// Verwendung der Presets: {attribute 'Preset.HochlaufzeitMin' := '@.tMinZeit'}
// oder dirket als Zahl: {attribute 'Preset.HochlaufzeitMin' := 'T#1M'}
// muss über der Instanz von ST_UniAntrAnstgParamAggrHF stehen
// mögliche Presets: 'Preset.HochlaufzeitMin', 'Preset.HochlaufzeitMax'
{attribute 'MaschPara.Margin' := '0 10 0 0'}	
{attribute 'MaschPara.Name' := 'Hochlaufphase 1 Zeit'}
{attribute 'MaschPara.Type' := 'min'}
{attribute 'MaschPara.Min' := 'Preset.HochlaufzeitMin'}
{attribute 'MaschPara.Max' := 'Preset.HochlaufzeitMax'}
{attribute 'MaschPara.Info' := 'Minuten je Hochlaufphase mit der Drehzahl aus fBetrZyklDrehz1'}
{attribute 'MaschPara.TreeViewLayer' := '-1'}
{attribute 'MaschPara.GroupName' := 'Preset.GroupName'}
	tBetrZyklPhase1	:TIME	:= T#1M;
// Verwendung der Presets: {attribute 'Preset.HochlaufzeitMin' := '@.tMinZeit'}
// oder dirket als Zahl: {attribute 'Preset.HochlaufzeitMin' := 'T#1M'}
// muss über der Instanz von ST_UniAntrAnstgParamAggrHF stehen
// mögliche Presets: 'Preset.HochlaufzeitMin', 'Preset.HochlaufzeitMax'
{attribute 'MaschPara.Name' := 'Hochlaufphase 2 Zeit'}
{attribute 'MaschPara.Type' := 'min'}
{attribute 'MaschPara.Min' := 'Preset.HochlaufzeitMin'}
{attribute 'MaschPara.Max' := 'Preset.HochlaufzeitMax'}
{attribute 'MaschPara.Info' := 'Minuten je Hochlaufphase mit der Drehzahl aus fBetrZyklDrehz2'}
{attribute 'MaschPara.TreeViewLayer' := '-1'}
{attribute 'MaschPara.GroupName' := 'Preset.GroupName'}
	tBetrZyklPhase2	:TIME	:= T#1M;
// Verwendung der Presets: {attribute 'Preset.HochlaufzeitMin' := '@.tMinZeit'}
// oder dirket als Zahl: {attribute 'Preset.HochlaufzeitMin' := 'T#1M'}
// muss über der Instanz von ST_UniAntrAnstgParamAggrHF stehen
// mögliche Presets: 'Preset.HochlaufzeitMin', 'Preset.HochlaufzeitMax'
{attribute 'MaschPara.Name' := 'Hochlaufphase 3 Zeit'}
{attribute 'MaschPara.Type' := 'min'}
{attribute 'MaschPara.Min' := 'Preset.HochlaufzeitMin'}
{attribute 'MaschPara.Max' := 'Preset.HochlaufzeitMax'}
{attribute 'MaschPara.Info' := 'Minuten je Hochlaufphase mit der Drehzahl aus fBetrZyklDrehz3'}
{attribute 'MaschPara.TreeViewLayer' := '-1'}
{attribute 'MaschPara.GroupName' := 'Preset.GroupName'}
	tBetrZyklPhase3	:TIME	:= T#1M;
// Verwendung der Presets: {attribute 'Preset.HochlaufzeitMin' := '@.tMinZeit'}
// oder dirket als Zahl: {attribute 'Preset.HochlaufzeitMin' := 'T#1M'}
// muss über der Instanz von ST_UniAntrAnstgParamAggrHF stehen
// mögliche Presets: 'Preset.HochlaufzeitMin', 'Preset.HochlaufzeitMax'
{attribute 'MaschPara.Name' := 'Hochlaufphase 4 Zeit'}
{attribute 'MaschPara.Type' := 'min'}
{attribute 'MaschPara.Min' := 'Preset.HochlaufzeitMin'}
{attribute 'MaschPara.Max' := 'Preset.HochlaufzeitMax'}
{attribute 'MaschPara.Info' := 'Minuten je Hochlaufphase mit der Drehzahl aus fBetrZyklDrehz4'}
{attribute 'MaschPara.TreeViewLayer' := '-1'}
{attribute 'MaschPara.GroupName' := 'Preset.GroupName'}
	tBetrZyklPhase4	:TIME	:= T#1M;
// Verwendung der Presets: {attribute 'Preset.StillstandMin' := '@.tMinZeit'}
// oder dirket als Zahl: {attribute 'Preset.StillstandMin' := 'T#1M'}
// muss über der Instanz von ST_UniAntrAnstgParamAggrHF stehen
// mögliche Presets: 'Preset.StillstandMin', 'Preset.StillstandMax'
{attribute 'MaschPara.Name' := 'Maximale Stillstandzeit'}
{attribute 'MaschPara.Type' := 'min'}
{attribute 'MaschPara.Min' := 'Preset.StillstandMin'}
{attribute 'MaschPara.Max' := 'Preset.StillstandMax'}
{attribute 'MaschPara.Info' := 'Zeit in Minuten bis eine neue Hochlaufphase notwendig wird'}
{attribute 'MaschPara.TreeViewLayer' := '-1'}
{attribute 'MaschPara.GroupName' := 'Preset.GroupName'}
	tMaxStillstandszeit	:TIME	:= T#15M;
// Verwendung der Presets: {attribute 'Preset.HochlaufdrehzMin' := '@.fMinDrehzahl'}
// oder dirket als Zahl: {attribute 'Preset.HochlaufdrehzMin' := '50'}
// muss über der Instanz von ST_UniAntrAnstgParamAggrHF stehen
// mögliche Presets: 'Preset.HochlaufdrehzMin', 'Preset.HochlaufdrehzMax'
{attribute 'MaschPara.Name' := 'Hochlaufphase 1 Drehzahl'}
{attribute 'MaschPara.Type' := '%'}
{attribute 'MaschPara.Min' := 'Preset.HochlaufdrehzMin'}
{attribute 'MaschPara.Max' := 'Preset.HochlaufdrehzMax'}
{attribute 'MaschPara.Info' := 'Prozentuale Drehzahl je Hochlaufphase'}	
{attribute 'MaschPara.TreeViewLayer' := '-1'}
{attribute 'MaschPara.GroupName' := 'Preset.GroupName'}
	fBetrZyklDrehz1	:LREAL := 50;
// Verwendung der Presets: {attribute 'Preset.HochlaufdrehzMin' := '@.fMinDrehzahl'}
// oder dirket als Zahl: {attribute 'Preset.HochlaufdrehzMin' := '75'}
// muss über der Instanz von ST_UniAntrAnstgParamAggrHF stehen
// mögliche Presets: 'Preset.HochlaufdrehzMin', 'Preset.HochlaufdrehzMax'
{attribute 'MaschPara.Name' := 'Hochlaufphase 2 Drehzahl'}
{attribute 'MaschPara.Type' := '%'}
{attribute 'MaschPara.Min' := 'Preset.HochlaufdrehzMin'}
{attribute 'MaschPara.Max' := 'Preset.HochlaufdrehzMax'}
{attribute 'MaschPara.Info' := 'Prozentuale Drehzahl je Hochlaufphase'}	
{attribute 'MaschPara.TreeViewLayer' := '-1'}
{attribute 'MaschPara.GroupName' := 'Preset.GroupName'}
	fBetrZyklDrehz2	:LREAL := 75;
// Verwendung der Presets: {attribute 'Preset.HochlaufdrehzMin' := '@.fMinDrehzahl'}
// oder dirket als Zahl: {attribute 'Preset.HochlaufdrehzMin' := '100'}
// muss über der Instanz von ST_UniAntrAnstgParamAggrHF stehen
// mögliche Presets: 'Preset.HochlaufdrehzMin', 'Preset.HochlaufdrehzMax'
{attribute 'MaschPara.Name' := 'Hochlaufphase 3 Drehzahl'}
{attribute 'MaschPara.Type' := '%'}
{attribute 'MaschPara.Min' := 'Preset.HochlaufdrehzMin'}
{attribute 'MaschPara.Max' := 'Preset.HochlaufdrehzMax'}
{attribute 'MaschPara.Info' := 'Prozentuale Drehzahl je Hochlaufphase'}	
{attribute 'MaschPara.TreeViewLayer' := '-1'}
{attribute 'MaschPara.GroupName' := 'Preset.GroupName'}
	fBetrZyklDrehz3	:LREAL := 100;
// Verwendung der Presets: {attribute 'Preset.HochlaufdrehzMin' := '@.fMinDrehzahl'}
// oder dirket als Zahl: {attribute 'Preset.HochlaufdrehzMin' := '20'}
// muss über der Instanz von ST_UniAntrAnstgParamAggrHF stehen
// mögliche Presets: 'Preset.HochlaufdrehzMin', 'Preset.HochlaufdrehzMax'
{attribute 'MaschPara.Name' := 'Hochlaufphase 4 Drehzahl'}
{attribute 'MaschPara.Type' := '%'}
{attribute 'MaschPara.Min' := 'Preset.HochlaufdrehzMin'}
{attribute 'MaschPara.Max' := 'Preset.HochlaufdrehzMax'}
{attribute 'MaschPara.Info' := 'Prozentuale Drehzahl je Hochlaufphase'}	
{attribute 'MaschPara.TreeViewLayer' := '-1'}
{attribute 'MaschPara.GroupName' := 'Preset.GroupName'}
	fBetrZyklDrehz4	:LREAL := 20;
	
END_STRUCT
END_TYPE

// DUTs/HMI_Parameter/ST_UniAntrAnstgParamTrsp
// Diese Struktur deklariert Parameter für den UniAnstgSEW-Baustein wenn dieser als Transport genutzt wird.
// Verwendung der Presets: {attribute 'Preset.GeschwMin' := '@.fMinGeschwindigkeitVMin'}
// oder dirket als Zahl: {attribute 'Preset.GeschwMin' := '10'}
// muss über der Instanz von ST_UniAntrAnstgParamTrsp stehen
// mögliche Presets: 'Preset.GeschwMin', 'Preset.GeschwMax'
// dazu kommt noch ein Preset für die Gruppierung der Parameter, also eine Überschrift.
// dieses wird so verwender: {attribute 'Preset.GroupName' := 'Hier ein Gruppenname'}
// der Gruppenname kann auch mit @.XXX eine globale Variable oder eine Variable in der folgenden Instantz der Struktur sein.
{attribute 'pack_mode' := '1'}
TYPE ST_UniAntrAnstgParamTrsp :
STRUCT
// Verwendung der Presets: {attribute 'Preset.GeschwMin' := '@.fMinGeschwindigkeitVMin'}
// oder dirket als Zahl: {attribute 'Preset.GeschwMin' := '10'}
// muss über der Instanz von ST_UniAntrAnstgParamTrsp stehen
// mögliche Presets: 'Preset.GeschwMin', 'Preset.GeschwMax'
//{attribute 'MaschPara.Margin' := '0 20 0 0'}	
{attribute 'MaschPara.Name' := 'minimale Geschwindigkeit'}
{attribute 'MaschPara.Type' := 'm/min'}
{attribute 'MaschPara.Min' := 'Preset.GeschwMin'}
{attribute 'MaschPara.Max' := 'Preset.GeschwMax'}
{attribute 'MaschPara.Info' := 'minimale Geschwindigkeit'}		
{attribute 'MaschPara.TreeViewLayer' := '-1'}
{attribute 'MaschPara.GroupName' := 'Preset.GroupName'}
	fVmin		:LREAL;
// Verwendung der Presets: {attribute 'Preset.GeschwMin' := '@.fMinGeschwindigkeitVMax'}
// oder dirket als Zahl: {attribute 'Preset.GeschwMin' := '10'}
// muss über der Instanz von ST_UniAntrAnstgParamTrsp stehen
// mögliche Presets: 'Preset.GeschwMin', 'Preset.GeschwMax'
{attribute 'MaschPara.Name' := 'maximale Geschwindigkeit'}
{attribute 'MaschPara.Type' := 'm/min'}
{attribute 'MaschPara.Min' := 'Preset.GeschwMin'}
{attribute 'MaschPara.Max' := 'Preset.GeschwMax'}
{attribute 'MaschPara.Info' := 'maximale Geschwindigkeit'}	
{attribute 'MaschPara.TreeViewLayer' := '-1'}
{attribute 'MaschPara.GroupName' := 'Preset.GroupName'}
	fVmax		:LREAL;
// Verwendung der Presets: {attribute 'Preset.GeschwMin' := '@.fMinGeschwindigkeitV1'}
// oder dirket als Zahl: {attribute 'Preset.GeschwMin' := '10'}
// muss über der Instanz von ST_UniAntrAnstgParamTrsp stehen
// mögliche Presets: 'Preset.GeschwMin', 'Preset.GeschwMax'
{attribute 'MaschPara.Name' := 'Geschwindigkeit 1'}
{attribute 'MaschPara.Type' := 'm/min'}
{attribute 'MaschPara.Min' := 'Preset.GeschwMin'}
{attribute 'MaschPara.Max' := 'Preset.GeschwMax'}
{attribute 'MaschPara.Info' := 'Geschwindigkeit 1'}
{attribute 'MaschPara.TreeViewLayer' := '-1'}
{attribute 'MaschPara.GroupName' := 'Preset.GroupName'}
	fV_1		:LREAL;	
// Verwendung der Presets: {attribute 'Preset.GeschwMin' := '@.fMinGeschwindigkeitV2'}
// oder dirket als Zahl: {attribute 'Preset.GeschwMin' := '10'}
// muss über der Instanz von ST_UniAntrAnstgParamTrsp stehen
// mögliche Presets: 'Preset.GeschwMin', 'Preset.GeschwMax'
{attribute 'MaschPara.Name' := 'Geschwindigkeit 2'}
{attribute 'MaschPara.Type' := 'm/min'}
{attribute 'MaschPara.Min' := 'Preset.GeschwMin'}
{attribute 'MaschPara.Max' := 'Preset.GeschwMax'}
{attribute 'MaschPara.Info' := 'Geschwindigkeit 2'}	
{attribute 'MaschPara.TreeViewLayer' := '-1'}
{attribute 'MaschPara.GroupName' := 'Preset.GroupName'}
	fV_2		:LREAL;	
// Verwendung der Presets: {attribute 'Preset.GeschwMin' := '@.fMinGeschwindigkeitV3'}
// oder dirket als Zahl: {attribute 'Preset.GeschwMin' := '10'}
// muss über der Instanz von ST_UniAntrAnstgParamTrsp stehen
// mögliche Presets: 'Preset.GeschwMin', 'Preset.GeschwMax'
{attribute 'MaschPara.Name' := 'Geschwindigkeit 3'}
{attribute 'MaschPara.Type' := 'm/min'}
{attribute 'MaschPara.Min' := 'Preset.GeschwMin'}
{attribute 'MaschPara.Max' := 'Preset.GeschwMax'}
{attribute 'MaschPara.Info' := 'Geschwindigkeit 3'}	
{attribute 'MaschPara.TreeViewLayer' := '-1'}
{attribute 'MaschPara.GroupName' := 'Preset.GroupName'}
	fV_3		:LREAL;
// Verwendung der Presets: {attribute 'Preset.RampeMin' := '@.fMinRampeAb'}
// oder dirket als Zahl: {attribute 'Preset.RampeMin' := '10'}
// muss über der Instanz von ST_UniAntrAnstgParamTrsp stehen
// mögliche Presets: 'Preset.RampeMin', 'Preset.RampeMax'
{attribute 'MaschPara.Name' := 'Verzögerungs-Rampe'}
{attribute 'MaschPara.Type' := 'ms'}
{attribute 'MaschPara.Min' := 'Preset.RampeMin'}
{attribute 'MaschPara.Max' := 'Preset.RampeMax'}
{attribute 'MaschPara.Info' := 'Verzögerungs-Rampe'}	
{attribute 'MaschPara.TreeViewLayer' := '-1'}
{attribute 'MaschPara.GroupName' := 'Preset.GroupName'}
	fRampe_ab:LREAL;
// Verwendung der Presets: {attribute 'Preset.RampeMin' := '@.fMinRampeAuf'}
// oder dirket als Zahl: {attribute 'Preset.RampeMin' := '10'}
// muss über der Instanz von ST_UniAntrAnstgParamTrsp stehen
// mögliche Presets: 'Preset.RampeMin', 'Preset.RampeMax'
{attribute 'MaschPara.Name' := 'Beschleunigungs-Rampe'}
{attribute 'MaschPara.Type' := 'ms'}
{attribute 'MaschPara.Min' := 'Preset.RampeMin'}
{attribute 'MaschPara.Max' := 'Preset.RampeMax'}
{attribute 'MaschPara.Info' := 'Beschleunigungs-Rampe'}	
{attribute 'MaschPara.TreeViewLayer' := '-1'}
{attribute 'MaschPara.GroupName' := 'Preset.GroupName'}
	fRampe_auf:LREAL;

END_STRUCT
END_TYPE

// DUTs/HMI_UniAnstgHandFktMeldungen/E_AnstgArtUniAktr
TYPE E_AnstgArtUniAktr :
(
	
	//Aktoransteuerung 0/1
	eAktrDef0Def1		:= 10,	// Es wird der String I_sInDef0 und I_sInDef1 genutzt
	eAktrEinAusschalt	:= 11,
	eAktrEinAusfahr	:= 12,
	eAktrHebenSenken	:= 13,
	//Aktoransteuerung 1/0
	eAktrDef1Def0		:= 20,	// Es wird der String I_sInDef0 und I_sInDef1 genutzt
	eAktrAusEinschalt	:= 21,
	eAktrAusEinfahr 	:= 22,
	eAktrSenkenHeben	:= 23
);
END_TYPE

// DUTs/HMI_UniAnstgHandFktMeldungen/E_AnstgArtUniAntr
// Definition der Uni-Antriebe
TYPE E_AnstgArtUniAntr :
(
	//Antriebsansteuerung 0/1
	eAntrDef0Def1		:= 10,	// Es wird der String I_sInDef0 und I_sInDef1 genutzt
	eAntrEinAusschalt	:= 11,
	eAntrEinAusfahr	:= 12,
	eAntrHebenSenken	:= 13,
	eAntrVorZurueck	:= 14,
	//Antriebsansteuerung 1/0
	eAntrDef1Def0		:= 50,	// Es wird der String I_sInDef0 und I_sInDef1 genutzt
	eAntrAusEinschalt	:= 51,
	eAntrAusEinfahr 	:= 52,
	eAntrSenkenHeben	:= 53,
	eAntrZurueckVor	:= 54
);
END_TYPE

// DUTs/HMI_UniAnstgHandFktMeldungen/E_AnstgArtUniWkzg
TYPE E_AnstgArtUniWkzg :
(
	// die Zahlen 0-8 sind reserviert um abwärtskompatiebel zu bleiben
	//Zylinderzuweisung 0/1
	eWkzgDef0Def1			:= 10,	// Es wird der String I_sInDef0 und I_sInDef1 genutzt
	eWkzgGrdArbstlg		:= 11,	// Taste 1: Arbeitsstellung Taste 2: Grundstellung
	eWkzgAbsAnheb			:= 12,	// Taste 1: absenken Taste 2: anheben
	eWkzgEinAusfahr		:= 13,	// Taste 1: einfahren Taste 2: ausfahren
	eWkzgZurVorfahr		:= 14,	// Taste 1: zurückfahren Taste 2: vorfahren
	eWkzgEinAussteun		:=	15,	// Taste 1: einsteuern Taste 2: aussteuern
	eWkzgLoesSpann			:= 16,	// Taste 1: lösen Taste 2: spannen
	eWkzgOeffnSchliess	:= 17,	// Taste 1: öffnen Taste 2: schließen
	eWkzgKlemLoesen		:= 18,	// Taste 1: lösen Taste 2: klemmen
	//Zylinderzuweisung 1/0
	eWkzgDef1Def0			:= 50,	// Es wird der String I_sInDef1 und I_sInDef0 genutzt
	eWkzgArbGrdstlg		:= 51,	// Taste 1: Arbeitsstellung Taste 2: Grundstellung
	eWkzgAnhAbsenk 		:= 52,	// Taste 1: anheben Taste 2: absenken
	eWkzgAusEinfahr		:= 53,	// Taste 1: ausfahren Taste 2: einfahren
	eWkzgVorZurfahr		:= 54,	// Taste 1: vorfahren Taste 2: zurückfahren
	eWkzgAusEinsteun		:=	55,	// Taste 1: aussteuern Taste 2: einsteuern
	eWkzgSpannLoes			:= 56,	// Taste 1: spannen Taste 2: lösen
	eWkzgSchliessOeffn	:= 57,	// Taste 1: schließen Taste 2: öffnen
	eWkzgLoesKlem			:= 58		// Taste 1: klemmen Taste 2: lösen
);
END_TYPE

// DUTs/HMI_UniAnstgHandFktMeldungen/E_AnstgArtUniZyli
TYPE E_AnstgArtUniZyli :
(
	//Zylinderzuweisung 0/1
	eZyliDef0Def1			:= 10,
	eZyliGrdArbstlg		:= 11,
	eZyliAbsAnheb			:= 12,
	eZyliEinAusfahr		:= 13,
	eZyliZurVorfahr		:= 14,
	eZyliEinAussteun		:=	15,
	eZyliLoesSpann			:= 16,
	eZyliOeffnSchliess	:= 18,
	eZyliZu0Zu180			:= 19,
	//Zylinderzuweisung 1/0
	eZyliDef1Def0			:= 50,
	eZyliArbGrdstlg		:= 51,
	eZyliAnhAbsenk			:= 52,
	eZyliAusEinfahr		:= 53,
	eZyliVorZurfahr		:= 54,
	eZyliAusEinsteun		:=	55,
	eZyliSpannLoes			:= 56,
	eZyliSchliessOeffn	:= 58,
	eZyliZu180Zu0			:= 59
);
END_TYPE

// DUTs/HMI_UniAnstgHandFktMeldungen/E_AntriebTyp
{attribute 'strict'}
TYPE E_AntriebTyp :
(
	eAggregat		:= 1,	//Antriebstyp 01: Ansteuerung als Bohraggregate etc.
	eTransport		:= 2,	//Antriebstyp 02: Ansteuerung als Transportsegmente etc.
	eVerstellg		:= 3,	//Antriebstyp 03: Ansteuerung als Schleichfahrt-Stopp-Verstellungen etc.
	eEilSchleich	:= 4,	//Antriebstyp 04: Ansteuerung als Eil/Schleich-Achse
	eAggregatHF		:= 5	//Antriebstyp 05: Ansteuerung als Hochfrequente Aggregate mit Warmlaufphase
);
END_TYPE

// DUTs/HMI_UniAnstgHandFktMeldungen/E_ZylinderTyp
{attribute 'strict'}
TYPE E_ZylinderTyp :
(	eZyliRueckstA1E0		:= 1,	// Zylindertyp 01: Anstg. 1 Rückstlg. /Abfrg.0
	eZyliRueckstA1E01		:= 2,	// Zylindertyp 02: Anstg. 1 Rückstlg. /Abfrg.0-1
	eZyliRueckstA01E0		:= 3,	// Zylindertyp 03: Anstg. 0-1 Rückstlg. /Abfrg.0
	eZyliRueckstA01E01	:= 4,	// Zylindertyp 04: Anstg. 0-1 Rückstlg. /Abfrg.0-1
	eZyliImpstlgA01E0		:= 5,	// Zylindertyp 05: Anstg. 0-1 Impulsstlg. /Abfrg.0
	eZyliImpstlgA01E01	:= 6,	// Zylindertyp 06: Anstg. 0-1 Impulsstlg. /Abfrg.0-1
	eZyliMittlstlgA01E01	:= 7	// Zylindertyp 07: Anstg. 0-1 Mittelstlg. /Abfrg.0-1
);
END_TYPE

// DUTs/HMI_UniAnstgHandFktMeldungen/ST_UniAchsAnstg
// Diese Struktur wird intern in dem Uni-Baustein FB_UniAchsAnstgNEU verwendet.
// Sie deklariert die Handfunktionen und Meldungen einer Achse.
{attribute 'pack_mode' := '1'}
TYPE ST_UniAchsAnstg :
STRUCT
	 
// Array von 5 Handfunktionen für die Steuerung einer Achse aus der HMI heraus.
// Taste 1: Achse negativ fahren
// Taste 2: Achse positiv fahren
// Taste 3: Platzhalter
// Taste 4: Platzhalter
// Taste 5: Reset
{attribute 'MaschPara.Name' := 'Handfunktion:'}	// Das Array ist Teil der Handfunktionen und wird mit 'Handfunktion:' betitelt
{attribute 'MaschPara.Handfunktion.Btn1' := '1 TextHandFkt'} // Handfunktion.Btn[X] ist der Taster im Array. TextHandFkt ist default Text, wenn z.B. die PLC nicht läuft
{attribute 'MaschPara.Handfunktion.Btn2' := '1 TextHandFkt'} // Handfunktion.Btn[X] ist der Taster im Array. TextHandFkt ist default Text, wenn z.B. die PLC nicht läuft
{attribute 'MaschPara.Handfunktion.Btn3' := '1 TextHandFkt'} // Handfunktion.Btn[X] ist der Taster im Array. TextHandFkt ist default Text, wenn z.B. die PLC nicht läuft
{attribute 'MaschPara.Handfunktion.Btn4' := '1 TextHandFkt'} // Handfunktion.Btn[X] ist der Taster im Array. TextHandFkt ist default Text, wenn z.B. die PLC nicht läuft
{attribute 'MaschPara.Handfunktion.Btn5' := '1 TextHandFkt'} // Handfunktion.Btn[X] ist der Taster im Array. TextHandFkt ist default Text, wenn z.B. die PLC nicht läuft
	stHandFktHMI	:ARRAY[1..5] OF ST_HandFktHMI;

// Fehlermeldungen aus dem FB_UniAchsAnstg	
{attribute 'Message.Struct'}	// Message.Struct bedeutet, dass die Strukur zu den Meldungen gehört und dem entsprechened von der HMI ausgelesen wird.
	stMeldAusgHMI		:ST_MeldTextUniAchs;

// Fehlermeldungen über die NcAchs-Struktur aus dem FB_AchsKontrlAnstg
{attribute 'Message.Struct'}	// Message.Struct bedeutet, dass die Strukur zu den Meldungen gehört und dem entsprechened von der HMI ausgelesen wird.
	stAchsMeldHMI		:ST_MeldAchsKontrl;
	
END_STRUCT
END_TYPE

// DUTs/HMI_UniAnstgHandFktMeldungen/ST_UniAktrAnstg
// Diese Struktur wird intern in dem Uni-Baustein FB_UniAktrAnstgNEU verwendet.
// Sie deklariert die Handfunktionen und Meldungen eines Aktors.
{attribute 'pack_mode' := '1'}
TYPE ST_UniAktrAnstg :
STRUCT
// Array von 2 Handfunktionen für die Steuerung eines Antriebes aus der HMI heraus.
// Taste 1: Text ist abhängig von der Funktion I_eAnstgDef
// Taste 2: Text ist abhängig von der Funktion I_eAnstgDef
{attribute 'MaschPara.Name' := 'Handfunktion:'}	// Das Array ist Teil der Handfunktionen und wird mit 'Handfunktion:' betitelt
{attribute 'MaschPara.Handfunktion.Btn1' := '1 TextHandFkt'} // Handfunktion.Btn[X] ist der Taster im Array. TextHandFkt ist default Text, wenn z.B. die PLC nicht läuft
{attribute 'MaschPara.Handfunktion.Btn2' := '1 TextHandFkt'} // Handfunktion.Btn[X] ist der Taster im Array. TextHandFkt ist default Text, wenn z.B. die PLC nicht läuft
	stHandFktHMI		:ARRAY[1..2] OF ST_HandFktHMI;	
// Meldungen eines Aktors
{attribute 'Message.Struct'}	// Message.Struct bedeutet, dass die Strukur zu den Meldungen gehört und dem entsprechened von der HMI ausgelesen wird.
	stMeldAusgHMI		:ST_MeldTextUniAktr;

END_STRUCT
END_TYPE

// DUTs/HMI_UniAnstgHandFktMeldungen/ST_UniAntrAnstg
// Diese Struktur wird intern in dem Uni-Baustein FB_UniAntrAnstgNEU verwendet.
// Sie deklariert die Handfunktionen und Meldungen eines Antriebes.
{attribute 'pack_mode' := '1'}
TYPE ST_UniAntrAnstg :
STRUCT
	 
{attribute 'MaschPara.Name' := 'Handfunktion:'}	// Das Array ist Teil der Handfunktionen und wird mit 'Handfunktion:' betitelt
{attribute 'MaschPara.Handfunktion.Btn1' := '1 TextHandFkt'} // Handfunktion.Btn[X] ist der Taster im Array. TextHandFkt ist default Text, wenn z.B. die PLC nicht läuft
{attribute 'MaschPara.Handfunktion.Btn2' := '1 TextHandFkt'} // Handfunktion.Btn[X] ist der Taster im Array. TextHandFkt ist default Text, wenn z.B. die PLC nicht läuft
{attribute 'MaschPara.Handfunktion.Btn3' := '1 TextHandFkt'} // Handfunktion.Btn[X] ist der Taster im Array. TextHandFkt ist default Text, wenn z.B. die PLC nicht läuft
{attribute 'MaschPara.Handfunktion.Btn4' := '1 TextHandFkt'} // Handfunktion.Btn[X] ist der Taster im Array. TextHandFkt ist default Text, wenn z.B. die PLC nicht läuft
{attribute 'MaschPara.Handfunktion.Btn5' := '1 TextHandFkt'} // Handfunktion.Btn[X] ist der Taster im Array. TextHandFkt ist default Text, wenn z.B. die PLC nicht läuft
	stHandFktHMI		:ARRAY[1..5] OF ST_HandFktHMI;

{attribute 'Message.Struct'}	// Message.Struct bedeutet, dass die Strukur zu den Meldungen gehört und dem entsprechened von der HMI ausgelesen wird.
	stMeldAusgHMI	:ST_MeldTextUniAntr;

END_STRUCT
END_TYPE

// DUTs/HMI_UniAnstgHandFktMeldungen/ST_UniBaustein
// Diese Struktur wird intern in den Uni-Bausteinen zur Adaption von alter HMI auf neue HMI verwendet.
{attribute 'pack_mode' := '1'}
TYPE ST_UniBaustein :
STRUCT

	bHandAnw0		:BOOL;
	bHandAnw1		:BOOL;
	bHandAnw2		:BOOL;
	bHandAnw3		:BOOL;
	nHandStat		:INT;	// .0/.1: grün .2/.3: rot .4:  .5: Zeile ausblenden .6/.7: sperren

	arrGrdstFkt		:ARRAY[0..3] OF BOOL;
	arrHandFkt		:ARRAY[0..3] OF BOOL;
	arrAutomFkt		:ARRAY[0..3] OF BOOL;
	arrFktAusfg		:ARRAY[0..3] OF BOOL;

END_STRUCT
END_TYPE

// DUTs/HMI_UniAnstgHandFktMeldungen/ST_UniGrdstlgAbl
// Struktur für eine standardisierte Grundstellungsanwahl mit einer HMI-Taste und Meldungen 
{attribute 'pack_mode' := '1'}
TYPE ST_UniGrdstlgAbl :
STRUCT
// Eine Handfunktionstaste für die Grundstellungsfahrt.
{attribute 'MaschPara.Name' := 'Handfunktion:'}	// Das Array ist Teil der Handfunktionen und wird mit 'Handfunktion:' betitelt
{attribute 'MaschPara.Handfunktion.Btn1' := '1 TextHandFkt'} // Handfunktion.Btn[X] ist der Taster im Array. TextHandFkt ist default Text, wenn z.B. die PLC nicht läuft
	stHandFktHMI		: ARRAY [1..1] OF ST_HandFktHMI;

// Meldungen für diese Grundstellungsfahrt.
{attribute 'Message.Struct'}	// Message.Struct bedeutet, dass die Strukur zu den Meldungen gehört und dem entsprechened von der HMI ausgelesen wird.
	stMeldAusgHMI		: ST_MeldGrundstellung;

END_STRUCT
END_TYPE

// DUTs/HMI_UniAnstgHandFktMeldungen/ST_UniWkzgAnstg
// Diese Struktur wird intern in dem Uni-Baustein FB_UniWkzgAnstgNEU verwendet.
// Sie deklariert die Handfunktionen irgendeines Werkzeuges.
{attribute 'pack_mode' := '1'}
TYPE ST_UniWkzgAnstg :
STRUCT
// Array von 2 Handfunktionen für die Steuerung eines Werkzeuges aus der HMI heraus.
// Taste 1: Text ist abhängig von der Funktion I_eAnstgDef
// Taste 2: Text ist abhängig von der Funktion I_eAnstgDef
{attribute 'MaschPara.Name' := 'Handfunktion:'}	// Das Array ist Teil der Handfunktionen und wird mit 'Handfunktion:' betitelt
{attribute 'MaschPara.Handfunktion.Btn1' := '1 TextHandFkt'} // Handfunktion.Btn[X] ist der Taster im Array. TextHandFkt ist default Text, wenn z.B. die PLC nicht läuft
{attribute 'MaschPara.Handfunktion.Btn2' := '1 TextHandFkt'} // Handfunktion.Btn[X] ist der Taster im Array. TextHandFkt ist default Text, wenn z.B. die PLC nicht läuft
	stHandFktHMI		:ARRAY[1..2] OF ST_HandFktHMI;	

{attribute 'Message.Struct'}	// Message.Struct bedeutet, dass die Strukur zu den Meldungen gehört und dem entsprechened von der HMI ausgelesen wird.
	stMeldAusgHMI		:ST_MeldTextUniWkzg;
END_STRUCT
END_TYPE

// DUTs/HMI_UniAnstgHandFktMeldungen/ST_UniZyliAnstg
// Diese Struktur wird intern in dem Uni-Baustein FB_UniZyliAnstg_TestMode verwendet.
// Sie deklariert die Handfunktionen und Meldungen eines Ventils mit Zylinders.
// Mit dieser Erweiterung für die Standardstruktur eines Zylinders kann ein Testmodus benutzt werden
{attribute 'pack_mode' := '1'}
TYPE ST_UniZyliAnstg :
STRUCT

{attribute 'MaschPara.Name' := 'Handfunktion:'}	// Das Array ist Teil der Handfunktionen und wird mit 'Handfunktion:' betitelt
{attribute 'MaschPara.Handfunktion.Btn1' := '1 TextHandFkt'} // Handfunktion.Btn[X] ist der Taster im Array. TextHandFkt ist default Text, wenn z.B. die PLC nicht läuft
{attribute 'MaschPara.Handfunktion.Btn2' := '1 TextHandFkt'} // Handfunktion.Btn[X] ist der Taster im Array. TextHandFkt ist default Text, wenn z.B. die PLC nicht läuft
{attribute 'MaschPara.Handfunktion.Btn3' := '1'} // Handfunktion.Btn[X] ist der Taster im Array. Hier kein Defaulttext, weil dadurch die Tasten ausgeblendet werden können
{attribute 'MaschPara.Handfunktion.Btn4' := '5'} // Handfunktion.Btn[X] ist der Taster im Array. Hier kein Defaulttext, weil dadurch die Tasten ausgeblendet werden können
{attribute 'MaschPara.Handfunktion.Btn5' := '1'} // Handfunktion.Btn[X] ist der Taster im Array. Hier kein Defaulttext, weil dadurch die Tasten ausgeblendet werden können
{attribute 'MaschPara.Handfunktion.Btn6' := '1'} // Handfunktion.Btn[X] ist der Taster im Array. Hier kein Defaulttext, weil dadurch die Tasten ausgeblendet werden können
	stHandFktHMI	:ARRAY[1..6] OF ST_HandFktHMI;

{attribute 'Message.Struct'}	// Message.Struct bedeutet, dass die Strukur zu den Meldungen gehört und dem entsprechened von der HMI ausgelesen wird.
	stMeldAusgHMI	:ST_MeldTextUniZyli;

END_STRUCT
END_TYPE

// DUTs/Meldebox/ST_MessageBox
{attribute 'pack_mode' := '1'}
// Diese Struktur muss zur Verwendung in einer Globalen Liste definiert werden und in den Einstellungen der HMI angegeben
// z.B. so: arrMessageBoxQueue : ARRAY[1..10] OF ST_MessageBox;
// TODO: muss in die BAAvalonLib wandern
TYPE ST_MessageBox :
STRUCT
	bShow				: BOOL;	// Boolsche Flanke die das Anzeigen der Meldungsbox auslöst. Flanke wird weggenommen, sobald eine Eingabe getätigt wurde.
	nResult			: INT;	// Ergebnis der Messagebox. 0 = keine Eingabe, 1 – 4 Nummer der ausgewählten Taste
	sInput			: STRING(255);	// Eingabe des Anwenders bei der InputMessageBox.
	nMode				: INT;	// Definiert, ob die MessageBox zur Eingabe dienen soll. 0 = Keine Eingabe 1 = Eingabe. Die Eingabe wird über sInput ausgelesen.
	sText				: STRING(255);	// Angezeigter Text.
	sMessageInfo	: STRING(255);	// Zusätzlicher Text, wenn ein Textfeld nicht reicht.
	sCaption			: STRING;	// Text in der Kopfzeile der MessageBox
	sButton1			: STRING(15);	// Text der 1. Taste (Leer = Taste unsichtbar)
	sButton2			: STRING(15);	// Text der 2. Taste (Leer = Taste unsichtbar)
	sButton3			: STRING(15);	// Text der 3. Taste (Leer = Taste unsichtbar)
	sButton4			: STRING(15);	// Text der 4. Taste (Leer = Taste unsichtbar)
	nIcon				: INT;	// Angezeigtes Bild 0 = Kein, 1 = Info, 2 = Warnung, 3 = Frage, 4 = Fehler
END_STRUCT
END_TYPE

// DUTs/NcAchsen/ST_AchsAuftrg
TYPE ST_AchsAuftrg :
STRUCT
	// Achs-Fahrauftrag
	sPTP_AuftrgTyp		:STRING(15);	// Beschreibung des Achstyp. Standard, Endlos oder Modulo
	
	bPTP_PosiFrg		:BOOL;	// Achse hat die Freigabe zu Positionieren. Betriebsbereit, beide Vorschubfreigaben und kein anderer Achsstart steht an.

	fPTP_ZielPos		:LREAL;	// aktuelle Zielposition für den Achsfahrauftrag
	fPTP_LetzZiel		:LREAL;	// Zu letzt angefahrene Zielposition
	fPTP_Geschw			:LREAL;	// in %
	ePTP_BuffMode		:MC_BufferMode;	(*MC_Aborting,
												  MC_Buffered,
												  MC_BlendingLow,
												  MC_BlendingPrevious,
												  MC_BlendingNext,
												  MC_BlendingHigh*)
	arrPTP_start		:ARRAY[1..3] OF BOOL;	// Achsstart für 3 verschiedene Betriebsmodi. Definiert in E_AchsFahrauftraege oder in NcParameter als Konstante
	bPTP_aktiv			:BOOL;	// Achsauftrag ist gestartet und auch aktiv
	bPTP_inZiel			:BOOL;	// Achsauftrag ist gestartet und im Ziel. Gibt es bei Endlosbetrieb nicht. Wird bei Verwendung vom FB_AchsStartAusf sofort wieder FALSE
	bPTP_inFenst		:BOOL;	// Achsauftrag ist gestartet und im Ziel +- 0.1 Grad oder mm. Gibt es bei Endlosbetrieb nicht.
	bPTP_stop			:BOOL;	// Achsauftrag wird gestoppt. Wird bei Verwendung vom FB_AchsStartAusf ggf. überschrieben
	bPTP_Autostop		:BOOL;	// wird aktuell nicht verwendet
	bPTP_gest			:BOOL;	// Achsauftrag wurde gestoppt. Ist nur bei aktivem bPTP_stop TRUE. Bedeutet, dass auch hier der FB_AchsStartAusf das überschreiben könnte
	bPTP_halt			:BOOL;	// Override auf 0%. Es wird mit der Beschleunigung aus dem Systemmanager gerampt
	bPTP_verz			:BOOL;	// Override auf den Wert aus der Freig-Struktur setzen.

END_STRUCT
END_TYPE

// DUTs/NcAchsen/ST_AchsFreigb
TYPE ST_AchsFreigb :
STRUCT
	// Achs-Freigaben
	{attribute 'hide'}
	bReglerFrg		:BOOL;	// intern. Wird durch die bAntrbEinFrg gesetzt.
	{attribute 'hide'}
	bVorsFrgNeg		:BOOL;	// intern. Wird durch bVorschFrg gesetzt, wenn die Endlage Negativ nicht angefahren wurde
	{attribute 'hide'}
	bVorsFrgPos		:BOOL;	// intern. Wird durch bVorschFrg gesetzt, wenn die Endlage Positiv nicht angefahren wurde
	
	fOverride		:LREAL	:= 10;	// Max-Override für diese Achse bei bPTP_verz
	
	bAntrbEinFrg	:BOOL;	// Schaltet die Reglerfreigabe und die Endlagenüberwachung ein
	bVorschFrg		:BOOL;	// Schaltet die Vorschubfreigabe mit einer internen Verzögerung (bReglerFrg+150ms) ein
	bSensEndlNeg	:BOOL;	// Externer Sensoreingang für die negative Endlage. Intern wird IQ_stAchse.stEinAusG.I_nDigitaleEingaenge.3 aus dem Bosch-Prozessdatenabbild verwendet
	bSensEndlPos	:BOOL;	// Externer Sensoreingang für die positive Endlage. Intern wird IQ_stAchse.stEinAusG.I_nDigitaleEingaenge.4 aus dem Bosch-Prozessdatenabbild verwendet
	bEndlFreifAkt	:BOOL;	// Vorschubfreigaben werden gesetzt und Hardwareendlagensensoren werden überschrieben um die Achse von diesen herunter zu fahren.
	bEndlgStop		:BOOL;	// Achse wurde auf einem Hardwareendlagensensor gestoppt und nicht zum Freifahren angewählt.
END_STRUCT
END_TYPE

// DUTs/NcAchsen/ST_AchsGrdfkt
TYPE ST_AchsGrdfkt :
STRUCT
	// Achs-Grundfunktion
	bRefrzSensor	:BOOL;	// Hardwaresensoreingang. Wird intern auf das ControlWord.5 geschrieben

	fIstSetzwert	:LREAL;	// Encoderwert auf den der Encoder gesetzt werden soll. Wird durch bIstw_setz angestoßen und bIstw_gesetz abgefragt.

	bRefrz_ausf		:BOOL;	// Referenzfahrt soll ausgeführt werden. Dafür muss die Vorschubfreigabe gesetzt sein.
	bRefrz_ausgf	:BOOL;	// Referenzfahrt wurde erfolgreich ausgeführt. Nur TRUE, wenn auch bRefrz_ausf TRUE ist
	bIstw_setz		:BOOL;	// Encoderwert wird absolut gesetzt. Reglerfreigabe muss dafür aus sein.
	bIstw_gesetz	:BOOL;	// Encoderwert wurde erfolgreich gesetzt. Nur TRUE, wenn bIstw_setz auch TRUE ist.
	bHdfkt_pos		:BOOL;	// Handfunktion (MC-Jog) positiv fahren. Nur mit Vorschubfreigabe. Wird von den Uni-Bausteinen beschrieben/überschrieben
	bHdfkt_neg		:BOOL;	// Handfunktion (MC-Jog) negativ fahren. Nur mit Vorschubfreigabe. Wird von den Uni-Bausteinen beschrieben/überschrieben
	bReset_ausf		:BOOL;	// NC-Reset wird ausgeführt. IQ_stAchse.stEinAusG.Q_nSignalsteuerwort.0 für Bosch-Servos wird beschrieben für einen Hardware-Reset.

END_STRUCT
END_TYPE

// DUTs/NcAchsen/ST_AchsInOut
{attribute 'pack_mode':='1'}
// Achsstruktur für Bosch-Rexroth-Servos
TYPE ST_AchsInOut :
STRUCT
	
	// Eingänge
	// #######################################################################
	I_nEinspeiseStatusword			AT %I*: WORD;	(*S-0-01720.0.2
										Bit 0 - 3 	-> reserviert
										Bit 4			-> Netzspannung OK
										Bit 5			-> Hardware bereit zum Einschalten
										Bit 6			-> Zwischenkreis wird gerade geladen, oder ist geladen
										Bit 8-9		-> Rückmeldung Betriebsart
										Bit 10		-> Zwischenkreisentladung angewählt und Zwischenkreis spannungsfrei (< ca. 35 V)
										Bit 11		-> Bremswiderstand aktiv
										Bit 12		-> Warnung aktiv
										Bit 13		-> Fehler aktiv
										Bit 14		-> Bereit zur Freigabe: Netzschütz geschlossen, Zwischenkreis geladen. Die versorgten Achsen zeigen "bb".
										Bit 15		-> Die Freigabe ist gegeben, d.h. der Zwischenkreis ist belastbar. Die versorgten Achsen können nach "Ab" geschaltet werden und die Antriebsfreigabe kann gesetzt werden.
															Bei den Wechselrichtern XM* muss das Bit von der Steuerung beschrieben werden, wenn der Versorger bzw. der versorgenden Umrichter den Status "Freigabe" gesetzt hat.
										*)

	I_nDCStatusword					AT %I*: WORD;	(*P-0-0115
										Bit 0 	 	-> Antrieb Betriebsbereit
										Bit 1			-> Antrieb bereit zur Leistungsabgabe
										Bit 2			-> Warnung (ZKL 2) steht an
										Bit 3			-> Antrieb folgt (ext.) Sollwertvorgabe
										Bit 4			-> Antrieb-Halt ist aktiv und Achse ist im Stillstand
										Bit 5			-> Kommandozustand hat sich geändert
										Bit 6			-> Antrieb folgt (int.) Sollwertvorgabe der SPS
										Bit 7			-> Haupt- oder Nebenbetriebsart aktiv und Initialisierung abgeschlossen, sonst 0
										Bit 8-11		-> Istbetriebsart 
										Bit 12		-> Antrieb hat Sollwertvorgabe erreicht. (Die Bildung des Bit abhängig von der aktiven BA ist weiter unten beschrieben).
										Bit 13		-> Antriebsfehler
										Bit 14/15	-> 00: Steuer- / Leistungsteil nicht betriebsbereit z.B. Antriebsfehler oder Phase 2)
															01: Steuerteil betriebsbereit (bb)
															10: Steuer- und Leistungsteil betriebsbereit (Ab)
															11: Antrieb momentenbehaftet (AF)

										*)

	I_nDigitaleEingaenge				AT %I*: DWORD;	// Hardwareeingänge von Bosch-Rexroth. Bit .3 und .4 sind die Hardwareendlagen 
	I_nStatusHaltebremse				AT %I*: WORD;	
	I_nStatusGehaltNennmoment		AT %I*: WORD;
	I_nBetriebsstundenzaehler		AT %I*: UDINT;
	I_nDiagnoseNummer					AT %I*: DWORD;
	
	I_nDrehmomentIstwert				AT %I*: INT;	// In 0,1%. Also 1000 ist 100%
	
	I_nSignalstatuswort				AT %I*: WORD;
	
	I_nZustandsklasse3				AT %I*: WORD;
	
	// Ausgänge
	// #######################################################################
	Q_nDrehmomentGrenzwert 			AT %Q*: INT;	// Drehmoment Grenzwert Bipolar in 0,1%. Also 1000 ist 100%

	Q_nEinspeiseSteuerwort			AT %Q*: WORD;	(*S-0-01720.0.1
										Bit 0 - 7 	-> reserviert
										Bit 8-9		-> Betriebsartvorwahl
										Bit 10		-> Funktion Zwischenkreisentladung starten
										Bit 11		-> n.v.
										Bit 12		-> Betätigung des versorgerintegrierten Betriebsbereitrelais, mit dem ein optionales Hauptschütz (vorgelagertes, zusätzliches Schaltelement) freigegeben werden kann.
										Bit 13		-> Fehler aktiv
										Bit 14		-> Zwischenkreis laden und Netzschütz einschalteten - Gerät geht in Gleichrichterbetrieb
										Bit 15		-> Freigabe, Sollbetriebsart aktivieren -> Wirkt auf die IGBT-Brücke des Versorgungsgeräts, aktiviert die DC-Zwischenkreisspannungsregelung und die Sollbetriebsart
										*)

	Q_nDCPowerControl					AT %Q*: WORD;	(*S-0-0240
										Bit 0 		->Der Zwischenkreis ist bereit zur Leistungsabgabe und -aufnahme (Achse meldet antriebsbereit "Ab")
										*)

	Q_nSignalsteuerwort				AT %Q*: WORD;	(*
										Bit 0 - ReglerReset,
										Bit 1 - Fahren auf Festanschlag
										Bit 2 - Bremsentest ausführen
										*)
	
	{attribute 'TcContextName':='Task_AchsFastStop'}
	Q_bAchsNcAchsFastStop			AT %Q*: BOOL;	// Vorschlag für eine Variable verbunden mit dem Faststop aus der NC. Diese Variable hat den TcContextName: 'Task_AchsFastStop'. Dafür muss diese Task mit diesem Namen natürlich existieren.

END_STRUCT
END_TYPE

// DUTs/NcAchsen/ST_AchsKoppln
TYPE ST_AchsKoppln :
STRUCT
	// Achs-Koppelfunktionen
	bAnkoppln		:BOOL;	// Achse an den Master nKopplMaster ankoppeln
	bAngekoplt		:BOOL;	// Achse ist angekoppelt. Ist TRUE, so lange bAnkoppln TRUE ist
	bAbkoppln		:BOOL;	// Achse abkoppeln
	bAbgekoplt		:BOOL;	//	Achse ist abgekoppelt. Ist TRUE, so lange bAbkoppln TRUE ist
	nKopplMaster	:INT;		// Masterachse für das bAnkoppln
	fKopplFakt		:LREAL;	// GearRatio im Verhältnis zum Master (nKopplMaster)
	nKopplStat		:DWORD;	// 0=Single/1=Master/2=Master-Slave/3=Slave aus IQ_fbAxisRef.NcToPlc.CoupleState

	fKorrektPos		:LREAL;	//Mittelwert (Achsen Mechanisch verbunden)
END_STRUCT
END_TYPE

// DUTs/NcAchsen/ST_AchsMeldg
{attribute 'hide'}
// Alles interne Meldestrukturen
TYPE ST_AchsMeldg :
STRUCT
	// Achs-Meldungen
{attribute 'hide'}
	bAntrbFehl		:BOOL;	// Reglerfreigabe gesetzt, aber nicht Betriebsbereit für 5s. Wird im AchsKtrlBaustein beschrieben und im UniBaustein in die Meldestruktur ausgegeben
{attribute 'hide'}
	bIstPosFehl		:BOOL;	// Achse steht außerhalb der Softwareendlage (+-5 mm oder Grad), ist referenziert und Softwareendlagen sind aktiv. Wird im AchsKtrlBaustein beschrieben und im UniBaustein in die Meldestruktur ausgegeben
{attribute 'hide'}
	bZielPosFehl	:BOOL;	// Achszielposition liegt ausßerhalb der Softwareendlage. Wird im AchsKtrlBaustein beschrieben und im UniBaustein in die Meldestruktur ausgegeben
{attribute 'hide'}
	bLfZeitFehl		:BOOL;	// Achse wurde gestartet, nicht in Ziel, Halt oder Stop für 60s. Wird im AchsKtrlBaustein beschrieben und im UniBaustein in die Meldestruktur ausgegeben

{attribute 'hide'}
	bEndlNegAngf	:BOOL;	// Endlage negativ wurde angefahren. Wird im AchsKtrlBaustein beschrieben und im UniBaustein in die Meldestruktur ausgegeben
{attribute 'hide'}
	bEndlPosAngf	:BOOL;	// Endlage positiv wurde angefahren. Wird im AchsKtrlBaustein beschrieben und im UniBaustein in die Meldestruktur ausgegeben

END_STRUCT
END_TYPE

// DUTs/NcAchsen/ST_AchsParam
TYPE ST_AchsParam :
STRUCT
	// Achs-Parameter

	bLesSchrFrg		:BOOL;	// bei steigender Flanke werden alle Parameter gelesen und geschrieben

	bOhnSoftEndl	:BOOL;	// Softwareendlagen werden bei der Zielposition nicht überwacht.

	fSoftEndlMin	:LREAL;	// RO aktuelle Softwareendlage
	fSoftEndlMax	:LREAL;	// RO aktuelle Softwareendlage
	bSoftEndlAkt	:BOOL;	// RO Softwareendlagen sind nicht aktiv
	fEilgGeschw		:LREAL;	// RO Maximale Achsgeschwindigkeit. In mm oder ° Nicht in %

	fEndlBegrMin	:LREAL;	// WO Softwareendlage min setzen
	fEndlBegrMax	:LREAL;	// WO Softwareendlage max setzen

	fPosVerrWert	:LREAL;	// Maschinen-Parameter. Wird auf die Zielposition aufaddiert. Das gleiche wie fPosOffsWert
	fPosOffsWert	:LREAL;	// Maschinen-Parameter. Wird auf die Zielposition aufaddiert. Das gleiche wie fPosVerrWert
	fGrdstlgPos		:LREAL;	// Maschinen-Parameter. Feste Zielposition bei dem Fahrauftrag arrPTP_start[cGrundPos]
	fGeschwVorg		:LREAL;	// Maschinen-Parameter. Geschwindigkeit beim Bremse einschleifen und als Zwischenspeicher zu verwenden. Bei Fahraufträgen im AchsKtrlBaustein wird immer fPTP_Geschw genommen
	fParkPos			:LREAL;	// Maschinen-Parameter. Nur ein Zwischenspeicher.

END_STRUCT
END_TYPE

// DUTs/NcAchsen/ST_AchsStatus
TYPE ST_AchsStatus :
STRUCT
	// Achs-Status
	bInReferz		:BOOL;	// RO Achse ist referenziert. Vorallem bei Eilschleichachsen wichtig. (direkt aus AXISREF.Status.Homed)
	bInStillst		:BOOL;	// RO Achse steht. (direkt aus AXISREF.Status.NotMoving)
	bFahrbewAkt		:BOOL;	// RO Achse wird bewegt (Encoder) oder bewegt sich selbst (Servo). (direkt aus AXISREF.Status.Moving)
	bFaehrtPos		:BOOL;	// RO Achse wird bewegt (Encoder) oder bewegt sich selbst (Servo) positiv. (direkt aus AXISREF.Status.PositiveDirection)
	bFaehrtNeg		:BOOL;	// RO Achse wird bewegt (Encoder) oder bewegt sich selbst (Servo) negativ. (direkt aus AXISREF.Status.NegativeDirection)
	bKonstFahrt		:BOOL;	// RO Achse hat eine konstante Geschwindigkeit erreicht. (direkt aus AXISREF.Status.ConstantVelocity)
	bZielPosErr		:BOOL;	// RO Achse hat ihre Zielposition erreicht. (Genauigkeit im Systemmanager angegeben) (direkt aus AXISREF.Status.InTargetPosition)
	bZielBerErr		:BOOL;	// RO Achse hat ihr Zielfenster erreicht. (Genauigkeit im Systemmanager angegeben) (direkt aus AXISREF.Status.InPositionArea)
	
	bInGrundPos		:BOOL;	// WO Achse in Grundstellung. Muss selbst beschrieben werden

	// Hardware-Status
	bAchseBTB		:BOOL;	// RO Umrichterstatus. Wird im UniAchsAnstg, UniAntrAnstgSEW oder CtrlXGrupEinschalt gesetzt.
	bFrgSchutzBer	:BOOL;	// WO Schutzbereich für diese Achse ist freigegeben. Wichtig für Ausgabe der Hardware-Fehler

END_STRUCT
END_TYPE

// DUTs/NcAchsen/ST_NcAchsen
// Achsstruktur für den FB_AchsKontrlAnstg
TYPE ST_NcAchsen:
STRUCT
	nAxNr				:INT;	// RO Achsnummer im Systemmanager
	sAxName			:STRING(31);	// RO NC-Achsname aus dem Systemmanager

	bNcFehler		:BOOL;	// RO NC hat einen Fehler
	nFehlerNr		:UDINT;	// RO NC Fehlernummer
	bBetrbBer		:BOOL;	// RO NC-Achse ist Betriebsbereit. Quasi das Häckchen. (direkt aus AXISREF.Status.Operational)
	bHwFehler		:BOOL;	// RO Umrichter ist nach Freigabe des Schutzbereiches für 5s nicht Betriebsbereit.

	fPosIstwert		:LREAL;	// RO Aktuelle Position (direkt aus AXISREF.NcToPlc.ActPos)
	fVeloIstwert	:LREAL;	// RO Aktuelle Geschwindigkeit (direkt aus AXISREF.NcToPlc.ActVelo)
	fModIstwert		:LREAL;	// RO Aktueller Modulowert (direkt aus AXISREF.NcToPlc.ModuloActPos)

	fAuftrOverride	:LREAL;	// RO Aktueller Override für den Fahrauftrag

	stStatus			:ST_AchsStatus;	// Achs-Status
	stParam			:ST_AchsParam;		// Achs-Parameter
	stFreigb			:ST_AchsFreigb;	// Achs-Freigaben
	stGrdfkt			:ST_AchsGrdfkt;	// Achs-Grundfunktionen
	stKoppln			:ST_AchsKoppln;	// Achs-Koppelfunktionen
	stAuftrg			:ST_AchsAuftrg;	// Achs-Fahrauftrag
	stMeldg			:ST_AchsMeldg;		// Achs-Meldungen
	
	stEinAusG		:ST_AchsInOut;		// Achs Ein- und Ausgangsstruktur für Bosch-Rexroth-Servos

END_STRUCT
END_TYPE

// DUTs/SEW/ST_SEWInput
{attribute 'pack_mode' := '1'}
TYPE ST_SEWInput :
STRUCT

	arrPI	:ARRAY[1..3] OF WORD;	// [1]: Status, [2]: Ist-Geschwindigkeit in %, [3]: Ist-Strom

END_STRUCT
END_TYPE

// DUTs/SEW/ST_SEWOutput
{attribute 'pack_mode' := '1'}
TYPE ST_SEWOutput :
STRUCT

	arrPO	:ARRAY[1..3] OF WORD;	// [1]: Steuerung, [2]: Soll-Geschwindigkeit, [3]: Rampe

END_STRUCT
END_TYPE

// DUTs/TwinSAFE/E_SafetyType
{attribute 'qualified_only'}
{attribute 'strict'}
TYPE E_SafetyType :
(
	eEL6900 := 1,
	eEL6910,
	eEL1904,
	eEL1918,
	eEL2904,
	eEL2911,
	eEL2912,
	eAX5805,
	eAX5806,
	eEK1914,
	eEP1908,
	eEP1918,
	eEP1957,
	eEP2918
);
END_TYPE

// DUTs/TwinSAFE/ST_TwinSAFE_Conn_Info
{attribute 'pack_mode' := '1'}
// Mit einer gemeinsamen Basis für alle Connections
TYPE ST_TwinSAFE_Conn_Info
EXTENDS ST_TwinSAFE_ConnInfoBasis:
STRUCT
	nInput	: BYTE;
	nOutput	: BYTE;
END_STRUCT
END_TYPE

// DUTs/TwinSAFE/ST_TwinSAFE_ConnInfoBasis
{attribute 'pack_mode' := '1'}
// Diese Struktur dient als Basis für alle Info-Strukturen die mit dem TwinSAFE verknüpft sind.
// Im Regelfall sind nur diese beiden Variablen (State und Diag) interessant.
// Wenn alle weiteren Strukturen auf dieser Basis basieren, kann jede erweiterte Struktur, egal wie viele Variablen hinzugekommen sind, an einen Eingang mit diesem Basistyp angelegt werden.
// Beispiel: Die Connections können verschiedene Ein- und Ausgänge haben. 1904 1Byte Eingang und 1Byte Ausgang und 1918 2Byte Eingang und 1 Byte Ausgang.
// Wenn beide Connection-Strukturen auf dieser Struktur basieren, können sie an einen Auswertbaustein angelegt werden. Es ist kein weiterer Baustein notwendig.
TYPE ST_TwinSAFE_ConnInfoBasis :
STRUCT
	nMapState	: USINT;	// State von TwinSAFE-Entität. Kann von einer Connection, Gruppe oder FB sein
	nMapDiag		: USINT;	// Diag von TwinSAFE-Entität. Kann von einer Connection, Gruppe oder FB sein
END_STRUCT
END_TYPE

// DUTs/TwinSAFE/ST_TwinSAFE_FB_Info
{attribute 'pack_mode' := '1'}
TYPE ST_TwinSAFE_FB_Info :
STRUCT
	nMapState		:USINT;
	nMapDiag			:UINT;
END_STRUCT
END_TYPE

// DUTs/TwinSAFE/ST_TwinSAFE_Group_Info
{attribute 'pack_mode' := '1'}
TYPE ST_TwinSAFE_Group_Info :
STRUCT

	nMapState			:USINT;
	nMapDiag				:USINT;

END_STRUCT
END_TYPE

// DUTs/TwinSAFE/ST_TwinSAFEConnInfo4Byte
{attribute 'pack_mode' := '1'}
// Mit einer gemeinsamen Basis für alle Connections
TYPE ST_TwinSAFEConnInfo4Byte
EXTENDS ST_TwinSAFE_ConnInfoBasis:
STRUCT
	nInput	: BYTE;
	nOutput	: BYTE;
END_STRUCT
END_TYPE

// DUTs/TwinSAFE/ST_TwinSAFEConnInfo5Byte
{attribute 'pack_mode' := '1'}
// Mit einer gemeinsamen Basis für alle Connections
TYPE ST_TwinSAFEConnInfo5Byte
EXTENDS ST_TwinSAFE_ConnInfoBasis:
STRUCT
	nInput1	: BYTE;
	nInput2	: BYTE;
	nOutput	: BYTE;
END_STRUCT
END_TYPE

// DUTs/TwinSAFE/ST_TwinSAFEKlemmenInfo
{attribute 'pack_mode' := '1'}
// Struktur für den Baustein FB_TwinSAFEKlemmeInfo.
TYPE ST_TwinSAFEKlemmenInfo :
STRUCT
	 nAdresse		: UINT;		// EtherCAT-Adresse
	 eTyp				: E_SafetyType;	// Typ der Safetyklemme
	 sName			: STRING;	// Name der Klemme im System Manager
	 nAnzFehler		: INT;		// Anzahl der anstehenden Fehler
	 arrFehlertext	: ARRAY [0..10] OF Tc2_System.T_MaxString;
	 arrFehler		: ARRAY [0..10] OF BOOL;
END_STRUCT
END_TYPE

// DUTs/ST_TimeStamp
{attribute 'pack_mode' := '1'}
// Diese Struktur muss durch den Functionsblock FB_Zeitstempel beschrieben werden
TYPE ST_TimeStamp :
STRUCT
	sQ					: STRING;	// Zeitstempel
	nStunde			: WORD;		// Stunde als Dezimalwert
	nMinute			: WORD;		// Minute als Dezimalwert
	nSekunde			: WORD;		// Sekunde als Dezimalwert
	nMilliSekunde	: WORD;		// Millisekungen als Dezimalwert
	nTag				: WORD;		// Tag als Dezimalwert
	nMonat			: WORD;		// Monat als Dezimalwert
	nJahr				: WORD;		// Jahr als Dezimalwert
	nTagDerWoche	: WORD;		// Tag der Woche  als Dezimalwert
END_STRUCT
END_TYPE

// DUTs/ST_TimeStruct
{attribute 'pack_mode' := '1'}
// Diese Struktur erweitert den standard Timestruct um ein String für den Zeitstempel.
// Dieser String muss durch die Function F_TimeStamp beschrieben werden
TYPE ST_TimeStruct EXTENDS Tc2_Utilities.TIMESTRUCT :
STRUCT
	sTimeStamp	:	STRING;	// String-Zeitstempel aus den Werten des TIMESTRUCT
END_STRUCT
END_TYPE

// POUs/ComPort_3_0_1_0/ST_MeldComPort
{attribute 'pack_mode' := '1'}
TYPE ST_MeldComPort :
STRUCT
{attribute 'Message.SourceID'}
	SourceID			:DINT;
	
{attribute 'Message.SourceName'}
   SourceName		:STRING	:= 'ComPort';
	
{attribute 'Message.Text' := 'Comport wurde noch nicht durch die SPS-Konfiguriert.'}
{attribute 'Message.Info' := ''}
{attribute 'Message.Type' := '1'}	
{attribute 'Message.Log'  := '0'}
	bMeldConfig		:BOOL;	// Comport nicht durch SPS konfiguriert
	
{attribute 'Message.Text' := 'Für den Comport wurden nicht alle Ein-/Ausgänge verknüpft.'}
{attribute 'Message.Info' := ''}
{attribute 'Message.Type' := '2'}	
{attribute 'Message.Log'  := '0'}
	bMeldMissingLink	:BOOL;	// Für den Comport wurden nicht alle Ein-/Ausgänge verknüpft

{attribute 'Message.Text' := 'Fehler beim Schreiben der Konfiguration auf die Klemme (CoE-Write-ErrorID: %Var1).'}
{attribute 'Message.Info' := ''}
{attribute 'Message.Type' := '5'}	
{attribute 'Message.Log'  := '1'}
{attribute 'Message.Var1' := 'nCoEWriteError'}
	bMeldConfigError	:BOOL;	// Fehler beim Schreiben der Konfiguration

{attribute 'Message.Text' := 'Fehler beim Empfangen von Daten (Recieve-ErrorID: %Var1).'}
{attribute 'Message.Info' := ''}
{attribute 'Message.Type' := '5'}	
{attribute 'Message.Log'  := '1'}
{attribute 'Message.Var1' := 'nRecieveError'}
	bMeldRecieveError	:BOOL;	// Fehler beim Empfangen von Daten

{attribute 'Message.Text' := 'Fehler beim Senden von Daten (Send-ErrorID: %Var1).'}
{attribute 'Message.Info' := ''}
{attribute 'Message.Type' := '5'}	
{attribute 'Message.Log'  := '1'}
{attribute 'Message.Var1' := 'nSendError'}
	bMeldSendError	:BOOL;	// Fehler beim Senden von Daten
	
{attribute 'Message.Text' := 'Timeout beim Empfangen von Daten (Timeoutzeit: %Var1 ms).'}
{attribute 'Message.Info' := ''}
{attribute 'Message.Type' := '5'}	
{attribute 'Message.Log'  := '1'}
{attribute 'Message.Var1' := 'tTimeoutZeit'}
	bMeldRecieveTimeout	:BOOL;	//  Timeout beim Empfangen von Daten

	nConfigError		:INT;	// Fehlernummer vom CoE-Write
	nRecieveError		:INT;	// Fehlernummer vom Recieve-FB
	nSendError			:INT;	// Fehlernummer vom Recieve-FB
	tTimeoutZeit		:TIME;	// Zeit beim Timeoutfehler
END_STRUCT
END_TYPE

// POUs/EtherCATDiagnose/E_EcCommState
{attribute 'to_string'}
TYPE E_EcCommState : (
	eEcState_UNDEFINED 	:= 0,
	eEcState_INIT 			:= 1,
	eEcState_PREOP 		:= 2,
	eEcState_BOOT 			:= 3,
	eEcState_SAFEOP 		:= 4,
	eEcState_OP 			:= 8
);
END_TYPE

// POUs/EtherCATDiagnose/ST_EcMasterDevState
{attribute 'pack_mode' := '1'}
TYPE ST_EcMasterDevState :
STRUCT
	eEcState	 				: E_EcCommState;
	nReserved				: ARRAY [0..2] OF UINT;

	bLinkError				: BOOL;
	bResetRequired			: BOOL;
	bMissFrmRedMode		: BOOL;
	bWatchdogTriggerd		: BOOL;
	bDriverNotFound		: BOOL;
	bResetActive			: BOOL;
	bAtLeastOneNotInOp	: BOOL;
	bDcNotInSync			: BOOL;
END_STRUCT
END_TYPE

// POUs/EtherCATDiagnose/ST_EcPortAddr
{attribute 'pack_mode' := '1'}
TYPE ST_EcPortAddr :
STRUCT
	nPortA : UINT;
	nPortB : UINT;
	nPortC : UINT;
	nPortD : UINT;
END_STRUCT
END_TYPE

// POUs/EtherCATDiagnose/ST_SlaveState
{attribute 'pack_mode' := '1'}
TYPE ST_SlaveState :
STRUCT
	// slave state
	eEcState 			: E_EcCommState;
	nReserved			: UINT;
	bError				: BOOL;
	bInvalidVPRS		: BOOL;
	nReserved2			: UINT;

	// link state
	bNoCommToSlave		: BOOL;
	bLinkError			: BOOL;
	bMissingLink		: BOOL;
	bUnexpectedLink	: BOOL;
	bPortA				: BOOL;
	bPortB				: BOOL;
	bPortC				: BOOL;
	bPortD				: BOOL;
END_STRUCT
END_TYPE

// POUs/EtherCATDiagnose/ST_SlaveStateInfo
{attribute 'pack_mode' := '1'}
TYPE ST_SlaveStateInfo :
STRUCT
	nIndex 				: DINT;
	sName 				: STRING; 		(* name of slave given in System Manager *)
	sType 				: STRING;		(* type of slave, e.g. EK1100*)
	nECAddr 				: UINT;			(* EtherCAT Slave Addr *)
	bDiagData			: BOOL;			(* DiagData in Slave State *)
	stPortCRCErrors	: ST_EcCrcErrorEx;(* Slave CRC-Errors, separate for each Port *)
	nSumCRCErrors		: UDINT;		(* Slave CRC-Errors, sum of all Ports *)
	stState 				: ST_SlaveState;(* EtherCAT State and Link state*)
END_STRUCT
END_TYPE

// POUs/EtherCATDiagnose/ST_SlaveStateInfoScanned
{attribute 'pack_mode' := '1'}
TYPE ST_SlaveStateInfoScanned :
STRUCT
	nIndex 			: DINT;
	sName 			: STRING; 		// Slavename von dem online erreichbaren Slave
	sType 			: STRING;		// Type des online erreichbaren Slaves, e.g. EK1100
	nECAddr 			: UINT;			// EtherCAT Slave Addresse
	bDifferentName	: BOOL;			// Name of Scanned configuration differs from Configured configuration
	bDifferentType	: BOOL;			// Type Of Scanned configuration differs from Configured configuration
	bDifferentAddr	: BOOL;			// EcAddress of Scanned configuration differs from Configured configuration
END_STRUCT
END_TYPE

// POUs/EtherCATDiagnose/ST_TopologyData
{attribute 'pack_mode' := '1'}
TYPE ST_TopologyData :
STRUCT
	nOwnPhysicalAddr 	: UINT;
	nOwnAutoIncAddr	: UINT;
	stPhysicalAddr		: ST_EcPortAddr;
	stAutoIncAddr		: ST_EcPortAddr;
	arrPortDelay		: ARRAY [0..2] OF UDINT;	// EC_AD, EC_DB, EC_BC
	arrReserved			: ARRAY [0..7] OF UDINT;
END_STRUCT
END_TYPE

// GVLs/AllgemeineParameter
{attribute 'Tc2GvlVarNames'}
VAR_GLOBAL CONSTANT
	cAnzSchutzBer		:INT:= 4;
	cAnzEinschGrp		:INT:= 3;
	
	// Meldearray-Definitionen im Schaltschrank
	cAnzKlimageraete		:INT:= 1;	// Anzahl der Klimageräte
	cAnzNetzteile			:INT:= 1;	// Anzahl der Netzteile
	cAnzSicherungen		:INT:= 1;	// Anzahl der Sicherungsautomaten. NICHT! die elektronischen Sicherungen.
	cAnzElekSicherungen	:INT:= 1;	// Anzahl der elektronischen Sicherungen.
	cAnzMSSchalter			:INT:= 0;	// Anzahl der Motorschutzschalter.
	cAnzThermoueberw		:INT:= 0;	// Anzahl der thermischen Überwachungen. Meist von Reglertrafos der Servo-Schrauber.
	cAnzWartungsEinheit	:INT:= 1;	// Anzahl der Wartungseinheiten für Betriebsdruck Meldungen.
	cAnzSonstige			:INT:= 0;	// Anzahl der sonstigen Meldungen.
	
	// Meldearray-Definitionen im Safety
	cAnzWartungstuer		:INT:= 1;	// Anzahl der Wartungstüren
	cAnzLichtgitter		:INT:= 0;	// Anzahl der Lichtgitter/Lichtschutzvorhänge
	cAnzNotHalt				:INT:= 8;	// Anzahl der NotHalt-Taster
	cAnzSafetyGruppen		:INT:= 5;	// Anzahl der Safetygruppen
	cAnzSafetyFBError		:INT:= 15;	// Anzahl der FB-Errors
	cAnzSafetyAusgaenge	:INT:= 10;	// Anzahl der Safetyausgänge
	cAnzSafetyKlemmen		:INT:= 20;	// Anzahl der Safetyklemmen für Diagnose
	cAnzSafetyConn4Byte	:INT:= 5;	// Anzahl der Ausgangsklemmen und alte Eingangsklemmen
	cAnzSafetyConn5Byte	:INT:= 10;	// Anzahl der Eingangsklemmen
	
	// EA-Aufbau
	cAnzEinspeis			:INT:= 5;	// Anzahl der Einspeisungen
	cAnzAuffrisch			:INT:= 5;	// Anzahl der Auffrischungen
	cAnzIOLinkKlemmen		:INT:= 5;	// Anzahl der IO-Linkklemmen
	cSlaveAddressArraySize	: UINT	:= 400;		(* Der Wert der Constanten iSLAVEADDR_ARR_SIZE
																	muß groesser/gleich Anzahl der EtherCAT-Teilnehmer sein.
																	Die Anzahl der EtherCAT-Teilnehmer steht in der Variablen 
																	nEcMasterSlaveCountCfg *)
	cMaxAnzahlSlaveError	: INT	:= 10;	// Anzahl der EtherCAT-Fehler, die angezeigt werden sollen.
	
	// EAP-Verbindungen
	cAnzEAPVerbindungen	:INT:= 2;	// Anzahl der Kommunikationsverbindungen mit anderen Anlagenteilen
	
	// ADS-Exchange
	cAnzKommError			:INT:= 5;	// Anzahl der Kommunikationsverbindungen mit anderen Anlagenteilen
	cAnzADS_EA_Error		:INT:= 5;	// Anzahl der EA-Exchangeverbindung zu anderen Anlagenteilen
	cAnzADS_Data_Error	:INT:= 5;	// Anzahl der Data-Exchangeverbindung zu anderen Anlagenteilen
	
	// Achsfehler
	cAnzAchsGruppen		:INT:= 0;	// Anzahl der Einspeisegruppen
END_VAR

// GVLs/ComPortParameterliste
{attribute 'Tc2GvlVarNames'}
VAR_GLOBAL CONSTANT
	cBufferSize_StringBuffer	: INT:=255;	(* Buffer beim String- und Barcodeempfang *)
	cBufferSize_IntBuffer		: INT:=300;	(* Buffer beim direkten und 4964R *)
	
	cAnzComports					: INT:= 0;	// Anzahl der seriellen Comports für RS232 
END_VAR

// GVLs/GlobalVar_Allgemein
{attribute 'Tc2GvlVarNames'}
VAR_GLOBAL
	(*Allgemein /Gesamtanlage*)
	bTaktLangsam				:BOOL;
	bTaktMittel					:BOOL;
	bTaktSchnell				:BOOL;
	bHinweistakt				:BOOL;

	bTakt2Langsam				:BOOL;
	bTakt2Mittel				:BOOL;
	bTakt2Schnell				:BOOL;
	bHinweistakt2				:BOOL;

	bPanelTastenAktiv			:BOOL;
	
	bFehlerEtherCATMaster		:BOOL;
	bFehlerEtherCATSlaveCount	:BOOL;
	bFehlerEtherCATAllg			:BOOL;
	bFehlerEtherCATSlave			:BOOL;
	
	(*Aktore und Ausgänge*)
	bVersEingAusgSchaltsOk	:BOOL;
	bVersEingAusgAnlagOk		:BOOL;
	
	bAnlagenStartBer1Ein		:BOOL;
	bAnlagenStartBer2Ein		:BOOL;
	bAnlagenStartBer3Ein		:BOOL;
	bAnlagenStartBer1VerzEin:BOOL;
	bAnlagenStartBer2VerzEin:BOOL;
	bAnlagenStartBer3VerzEin:BOOL;

	bVakPumpeAllgEin			:BOOL;

	bAntriebeAllg_Ein			:BOOL;

	bAntriebUmrGr1AchsFrg	:BOOL;
	bAntriebUmrGr2AchsFrg	:BOOL;
	bAntriebUmrGr3AchsFrg	:BOOL;
	
	(*Betriebsarten global*)
	bBetrartHand1Angew		:BOOL;
	bBetrartAutom1Angew		:BOOL;

	bBetrartHand2Angew		:BOOL;
	bBetrartAutom2Angew		:BOOL;

	bBetrartHand3Angew		:BOOL;
	bBetrartAutom3Angew		:BOOL;

	bModStepbetrAngew			:BOOL;
	bSteptaktAnlgBer1Ausf	:BOOL;
	bSteptaktAnlgBer2Ausf	:BOOL;
	bSteptaktAnlgBer3Ausf	:BOOL;
	
	bGrdstAnw_GesamtAnlage	:BOOL;
	bGrdstlgAblAllgAktiv		:BOOL;
	
	(*Schutzbereichspezifisch*)
	arrAusgGruppeFrg			:ARRAY[1..cAnzSchutzBer] OF BOOL;

	arrSchutzEinrGeschl		:ARRAY[1..cAnzSchutzBer] OF BOOL;
	arrSchutzEinrVerzGeschl	:ARRAY[1..cAnzSchutzBer] OF BOOL;

	arrAntrGruppe1Ein			:ARRAY[1..cAnzSchutzBer] OF BOOL;
	arrAntrGruppe2Ein			:ARRAY[1..cAnzSchutzBer] OF BOOL;
	arrAntrGruppe3Ein			:ARRAY[1..cAnzSchutzBer] OF BOOL;
	arrAntrGruppeFrg			:ARRAY[1..cAnzSchutzBer] OF BOOL;
	
	arrAchsGruppeFrg			:ARRAY[1..cAnzSchutzBer] OF BOOL;
	arrAchsGruppeFrgVerz		:ARRAY[1..cAnzSchutzBer] OF BOOL;
	
	arrBetrartAutomAktiv		:ARRAY[1..cAnzSchutzBer] OF BOOL;
	arrBetrartAutomSpeichn	:ARRAY[1..cAnzSchutzBer] OF BOOL;
	arrBetrartHandAktiv		:ARRAY[1..cAnzSchutzBer] OF BOOL;
	
	arrGrdstlgBetrAktiv		:ARRAY[1..cAnzSchutzBer] OF BOOL;
	
	arrGrdstAnw_GesamtBer	:ARRAY[1..cAnzSchutzBer] OF BOOL;
	
	arrAutoStopWartungsTuer	:ARRAY[1..cAnzSchutzBer] OF BOOL;
	arrTaktStopWartungsTuer	:ARRAY[1..cAnzSchutzBer] OF BOOL;
	arrTrspStopWartungsTuer	:ARRAY[1..cAnzSchutzBer] OF BOOL;

	arrEntrgAktWartungsTuer	:ARRAY[1..cAnzSchutzBer] OF BOOL;
	
	(**)
	bLeuchtmTest				:BOOL;	// Alle Meldeleuchten sollen leuchten

	bMeldTextAllgVorhand		:BOOL;	// eine Meldung ist vorhanden
	
	(*Zeiten*)
	sSystZeitDatum				:STRING(21);
	sSystZeitFuerLog			:STRING(21);

	(*Maschinenparameter*)
	bMaschParamAllgGueltig	:BOOL;	// Maschinenparameter von der HMI sind gültig

	(*Globaler Sensorfehler*)
	bSensFehlAllgVorhand		:BOOL;
		
	bIbnMaxDrehz				:BOOL;	// Bei allen SEW-Motoren die Drehzahl auf 100% einstellen
	
	bLuftdruckEin				:BOOL := TRUE;	// Druckluftventile ein. Im Normalfall bei TwinCAT aktiv
	
	stTimestamp					:ST_TimeStamp;
	stTimestruct				:ST_TimeStruct;
	
	bTwinSAFEInRun				: BOOL;
END_VAR

// GVLs/GlobalVar_Farben
{attribute 'Tc2GvlVarNames'}
// TODO: muss in die BAAvalonLib wandern

VAR_GLOBAL CONSTANT
	cDefault					:DWORD:= 16#00CCD3DA;	// Buttonfarbe, wenn nichts angewählt ist
	cOrange					:DWORD:= 16#F0FF6600;
	
	cDefaultAsString		:STRING:= '00CCD3DA';	// Buttonfarbe, wenn nichts angewählt ist
	cGruenAsString			:STRING:= 'F0719E47';
	cRotAsString			:STRING:= 'F0EF0000';
	cOrangeAsString		:STRING:= 'F0FF6600';
	cGelbAsString			:STRING:= 'F0FFCC00';
	cBlauAsString			:STRING:= 'F03A8DD1';
	cWeissAsString			:STRING:= 'F0FFFFFF';
	cGrauAsString			:STRING:= 'F0566B7E';
	
	// Aus der Doku der Avalon-HMI.
	// sDefaultString := TO_STRING(cDWORD) funktioniert übrigens nicht. Besser cDefaultAsString und ähnliches nutzen
	cSchwarz					:DWORD:= 16#00000000;	// FARBWERT
	cDunkelblau				:DWORD:= 16#F0000080;	// FARBWERT
	cDunkelgruen			:DWORD:= 16#F0008000;	// FARBWERT
	cDunkelcyan				:DWORD:= 16#E6008080;	// FARBWERT
	cDunkelrot				:DWORD:= 16#F0800000;	// FARBWERT
	cLila						:DWORD:= 16#F08000FF;	// FARBWERT
	cBraun					:DWORD:= 16#F0804000;	// FARBWERT
	cGrau						:DWORD:= 16#00C9D1CB;	// FARBWERT
	cDunkelgrau				:DWORD:= 16#00808080;	// FARBWERT
	cBlau						:DWORD:= 16#FF0000FF;	// FARBWERT
	cHellblau				:DWORD:= 16#AA0000FF;	// FARBWERT
	cGruen					:DWORD:= 16#F000FF00;	// FARBWERT
	cCcyan					:DWORD:= 16#F000FFFF;	// FARBWERT
	cRot						:DWORD:= 16#F0FF0000;	// FARBWERT
	cHellrot					:DWORD:= 16#AAFF0000;	// FARBWERT
	cPink						:DWORD:= 16#F0FF00FF;	// FARBWERT
	cGelb						:DWORD:= 16#F0FFFF00;	// FARBWERT
	cWeiss					:DWORD:= 16#00FFFFFF;	// FARBWERT
	cKEYBACK					:DWORD:= 16#26C8D0D7;	// FARBWERT
	
END_VAR

// GVLs/GlobalVar_TestMeld
{attribute 'Tc2GvlVarNames'}
VAR_GLOBAL
	bTestMeldAllgemein			: BOOL;	// Lib-intern nicht verwendet. Kann im Projekt für alles mögliche verwendet werden.
	bTestMeldAchs					: BOOL;	// Achse nicht Betriebsbereit testen
	bTestMeldAchsIstPosFehler	: BOOL;	// Achsen simulieren Ist-Position-Fehler
	bTestMeldAktr					: BOOL;	// alle Uni-Aktoren und Hydraulikaggregate melden einen Laufzeitfehler
	bTestMeldAntr					: BOOL;	// alle Uni-Antriebe Uni-SEW-Antriebe und Uni-SEW-IO-Anriebe melden nicht betriebsbereit
	bTestMeldAntrEilSchleich	: BOOL;	// alle Uni-SEW-Antriebe, die als Eil-Schleichachse definiert sind, melden nicht referenziert
	bTestMeldAntrVerstellg		: BOOL;	// alle Uni-SEW-Antriebe, die als Verstellantriebe definiert sind, melden nicht in Endlage
	bTestMeldAntrHF				: BOOL;	// alle Uni-SEW-Antriebe, die als Hochfrequenzantriebe definiert sind, melden Einlaufzyklus aktiv, beendet und Warmlaufzyklus aktiv
	bTestMeldGrdstlg				: BOOL;	// alle Uni-Grundstellungsbausteine melden Grundstellung aktiv, Fertig mit Entnahme und Fertig ohne Entnahme
	bTestMeldZyl					: BOOL;	// alle Uni-Zylinderbausteine melden nicht in Endlage, bzw. beide Endlagen aktiv
	
	bTestModeZylinder				: BOOL;	// in der HMI werden für alle Uni-Zylinder mit Testmodus auch die Testmodi angezeigt
END_VAR

// POUs/ComPort_2_0_1_0/F_ComReceiveBarcode
FUNCTION F_ComReceiveBarcode : ST_ComPortStringBuffer
VAR_INPUT
	I_pReceiveString	: POINTER TO ST_ComPortStringBuffer;
	I_pOptionsIntern	: POINTER TO ST_ComPortOptionsIntern;	// PLC - interne Schnittstellenparameter
END_VAR

VAR
	nStartPosition		: INT;
	nEndPosition		: INT;
	bPrefixFound		: BOOL;
END_VAR

F_ComReceiveBarcode.sData:='';

nStartPosition:=0;
IF 	I_pOptionsIntern^.nLenPrefix = 0 THEN
	bPrefixFound:=TRUE;
ELSE
	bPrefixFound:=FALSE;

	REPEAT
		nStartPosition:=FIND(I_pReceiveString^.sData,I_pOptionsIntern^.sPrefix);
		IF nStartPosition > 0 THEN
			bPrefixFound:=TRUE; (* Mindesten 1 x Prefix *)

			nStartPosition:=nStartPosition + I_pOptionsIntern^.nLenPrefix;
			I_pReceiveString^.sData:=MID(I_pReceiveString^.sData,LEN(I_pReceiveString^.sData)-nStartPosition+1,nStartPosition);
		END_IF
	UNTIL
		nStartPosition = 0
	END_REPEAT
END_IF

IF bPrefixFound = TRUE THEN
	nEndPosition:=0;

	IF I_pOptionsIntern^.nLenSuffix = 0 THEN
		nEndPosition:=LEN(I_pReceiveString^.sData);
	ELSE
		nEndPosition:=FIND(I_pReceiveString^.sData,I_pOptionsIntern^.sSuffix)-1;
	(*	IF EndPosition = 0 THEN
			EndPosition:=LEN(ReceiveString);
		END_IF
	*)
	END_IF

	IF nEndPosition > 0 THEN
		F_ComReceiveBarcode.sData:=MID(I_pReceiveString^.sData,nEndPosition,1);
	END_IF
END_IF

END_FUNCTION

// POUs/ComPort_2_0_1_0/F_ComSendBarcode
FUNCTION F_ComSendBarcode:ST_ComPortStringBuffer
VAR_INPUT
	I_pSendString				: POINTER TO ST_ComPortStringBuffer;
	I_pComPortOptionsIntern	: POINTER TO ST_ComPortOptionsIntern; 	(* PLC - interne Schnittstellenparameter *)
END_VAR

IF I_pComPortOptionsIntern^.nLenPrefix > 0 THEN
	F_ComSendBarcode.sData:=CONCAT(I_pComPortOptionsIntern^.sPrefix,I_pSendString^.sData);
ELSE
	F_ComSendBarcode:=I_pSendString^;
END_IF

IF I_pComPortOptionsIntern^.nLenSuffix > 0 THEN
	F_ComSendBarcode.sData:=CONCAT(F_ComSendBarcode.sData,I_pComPortOptionsIntern^.sSuffix);
END_IF

END_FUNCTION

// POUs/ComPort_2_0_1_0/FB_ComBackground
FUNCTION_BLOCK FB_ComBackground
VAR_INPUT
	I_pOptions		: POINTER TO ST_ComPortOptions;
	I_pComFlags		: POINTER TO ST_ComPortFlags;
END_VAR

VAR_IN_OUT
	IQ_stComPortIn		: ST_ComPortInData;
	IQ_stComPortOut	: ST_ComPortOutData;

	IQ_stRxBuffer		: Tc2_SerialCom.ComBuffer;	// Interner Empfangspuffer
	IQ_stTxBuffer		: Tc2_SerialCom.ComBuffer;	// Interner Sendepuffer
END_VAR

VAR
	fbPcComPortControl				: Tc2_SerialCom.SerialLineControl;
	fbKlemmeComPortControl3Bytes	: Tc2_SerialCom.SerialLineControl;
	fbKlemmeComPortControl5Bytes	: Tc2_SerialCom.SerialLineControl;
	fbKlemmeComPortControl22Bytes	: Tc2_SerialCom.SerialLineControl;
END_VAR

IF I_pOptions^.nAktiv = 1  AND I_pComFlags^.bConfigFlag = FALSE THEN
	CASE I_pOptions^.ePort OF
		E_ComPortHardware.cComportPc:
			fbPcComPortControl(
							Mode  := SERIALLINEMODE_PC_COM_PORT,
							pCOMin:=ADR(IQ_stComPortIn.stPCIn) ,
							pCOMout:=ADR(IQ_stComPortOut.stPCOut) ,
							SizeComIn := SIZEOF(IQ_stComPortIn.stPCIn),
							TxBuffer:=IQ_stTxBuffer ,
							RxBuffer:=IQ_stRxBuffer );

		E_ComPortHardware.cComportKL,E_ComPortHardware.cComportEL:
			CASE I_pOptions^.eComPortBytes OF
				E_ComPortKlemmenBytes.cComport3Bytes:
					fbKlemmeComPortControl3Bytes(
								Mode  := SERIALLINEMODE_KL6_3B_ALTERNATIVE,
								pCOMin:=ADR(IQ_stComPortIn.stKlemmeIn3B) ,
								pCOMout:=ADR(IQ_stComPortOut.stKlemmeOut3B) ,
								SizeComIn := SIZEOF(IQ_stComPortIn.stKlemmeIn3B),
								TxBuffer:=IQ_stTxBuffer ,
								RxBuffer:=IQ_stRxBuffer );

				E_ComPortKlemmenBytes.cComport5Bytes:
					fbKlemmeComPortControl5Bytes(
								Mode  := SERIALLINEMODE_KL6_5B_STANDARD,
								pCOMin:=ADR(IQ_stComPortIn.stKlemmeIn5B) ,
								pCOMout:=ADR(IQ_stComPortOut.stKlemmeOut5B) ,
								SizeComIn := SIZEOF(IQ_stComPortIn.stKlemmeIn5B),
								TxBuffer:=IQ_stTxBuffer ,
								RxBuffer:=IQ_stRxBuffer );

				E_ComPortKlemmenBytes.cComport22Bytes:
					fbKlemmeComPortControl22Bytes(
								Mode  := SERIALLINEMODE_KL6_22B_STANDARD,
								pCOMin:=ADR(IQ_stComPortIn.stKlemmeIn22B) ,
								pCOMout:=ADR(IQ_stComPortOut.stKlemmeOut22B) ,
								SizeComIn := SIZEOF(IQ_stComPortIn.stKlemmeIn22B),
								TxBuffer:=IQ_stTxBuffer ,
								RxBuffer:=IQ_stRxBuffer );
			END_CASE
	END_CASE;
END_IF

END_FUNCTION_BLOCK

// POUs/ComPort_2_0_1_0/FB_ComConfig
FUNCTION_BLOCK FB_ComConfig
VAR_INPUT
	I_pOptions				: POINTER TO ST_ComPortOptions;
END_VAR

VAR_OUTPUT
	Q_nConfigPortErrorId	: INT;
	Q_stOptionsIntern		: ST_ComPortOptionsIntern;
END_VAR

VAR_IN_OUT
	IQ_stComPortIn			: ST_ComPortInData;
	IQ_stComPortOut		: ST_ComPortOutData;

	IQ_stComFlags			: ST_ComPortFlags;
END_VAR

VAR
	bStartPLC				: BOOL;

	stComPortKL6configuration	: Tc2_SerialCom.KL6configuration;

	fbEcCoWrite				: FB_EcCoESdoWrite;
                     	
	nIndex					: WORD;
	nSubIndex				: BYTE;
                     	
	nWordBuffer				: WORD;
	bBuffer					: BOOL;
                     	
	nConfigState			: INT;
	nTmpVar					: UINT;
END_VAR

IF bStartPLC = FALSE THEN
	(* Initialisierung aller Schnittstellen nach Neustart und Reset *)
	IF I_pOptions^.nAktiv = 1  THEN
		IQ_stComFlags.bConfigFlag:=TRUE;
	END_IF
	bStartPLC:=TRUE;
END_IF

IF IQ_stComFlags.bConfigFlag = TRUE THEN
	CASE I_pOptions^.ePort OF
		E_ComPortHardware.cComportPc:
			IQ_stComFlags.bConfigFlag:=FALSE;

		E_ComPortHardware.cComportEL:
			CASE nConfigState OF
				0:  (* Baudrate *)
					nIndex:=16#4073;
					nSubIndex:=0;

					nWordBuffer:=4;
					nTmpVar:=I_pOptions^.nBaudrate;
					WHILE nTmpVar > 2400 DO
						nTmpVar:=nTmpVar/2;
						nWordBuffer:=nWordBuffer+1;
					END_WHILE

					fbEcCoWrite(
						sNetId:=F_CreateAmsNetId(IQ_stComPortIn.stInfoData.stADSNetId) ,
						nSlaveAddr:=IQ_stComPortIn.stInfoData.nADSPort,

						nSubIndex:=nSubIndex,
						nIndex:=nIndex,

						pSrcBuf:=ADR(nWordBuffer),
						cbBufLen:=SIZEOF(nWordBuffer),
						bExecute:=NOT fbEcCoWrite.bBusy,
						tTimeout:=T#3s);

				1:  (* Frame *)
					nIndex:=16#4074;
					nSubIndex:=0;

					IF I_pOptions^.nDatenbits = 7 THEN
						IF I_pOptions^.nStopbits = 1 THEN
							(*7x1 *)
							CASE I_pOptions^.nParitaet OF
								PARITY_NONE:nWordBuffer:=1;
								PARITY_EVEN:nWordBuffer:=1;
								PARITY_ODD:nWordBuffer:=2;
							END_CASE
						ELSE
							(*7x2 *)
							CASE I_pOptions^.nParitaet OF
								PARITY_NONE:nWordBuffer:=9;
								PARITY_EVEN:nWordBuffer:=9;
								PARITY_ODD:nWordBuffer:=10;
							END_CASE
						END_IF
					ELSE
						(*8x1 *)
						IF I_pOptions^.nStopbits = 1 THEN
							CASE I_pOptions^.nParitaet OF
								PARITY_NONE:nWordBuffer:=3;
								PARITY_EVEN:nWordBuffer:=4;
								PARITY_ODD:nWordBuffer:=5;
							END_CASE
						ELSE
							(*8x2 *)
							CASE I_pOptions^.nParitaet OF
								PARITY_NONE:nWordBuffer:=11;
								PARITY_EVEN:nWordBuffer:=12;
								PARITY_ODD:nWordBuffer:=13;
							END_CASE
						END_IF
					END_IF

					fbEcCoWrite(
						sNetId:=F_CreateAmsNetId(IQ_stComPortIn.stInfoData.stADSNetId) ,
						nSlaveAddr:=IQ_stComPortIn.stInfoData.nADSPort,

						nSubIndex:=nSubIndex,
						nIndex:=nIndex,

						pSrcBuf:=ADR(nWordBuffer),
						cbBufLen:=SIZEOF(nWordBuffer),
						bExecute:=NOT fbEcCoWrite.bBusy,
						tTimeout:=T#3s);

				2:  (* RTS/CTS *)
					nIndex:=16#4075;
					nSubIndex:=1;

					IF I_pOptions^.nHandshake = HANDSHAKE_RTSCTS THEN
						bBuffer:=TRUE;
					ELSE
						bBuffer:=FALSE;
					END_IF

					fbEcCoWrite(
						sNetId:=F_CreateAmsNetId(IQ_stComPortIn.stInfoData.stADSNetId) ,
						nSlaveAddr:=IQ_stComPortIn.stInfoData.nADSPort,

						nSubIndex:=nSubIndex,
						nIndex:=nIndex,

						pSrcBuf:=ADR(bBuffer),
						cbBufLen:=SIZEOF(bBuffer),
						bExecute:=NOT fbEcCoWrite.bBusy,
						tTimeout:=T#3s);

				3:  (* XON/XOFF tx *)
					nIndex:=16#4075;
					nSubIndex:=2;

					IF I_pOptions^.nHandshake = HANDSHAKE_XONXOFF THEN
						bBuffer:=TRUE;
					ELSE
						bBuffer:=FALSE;
					END_IF

					fbEcCoWrite(
						sNetId:=F_CreateAmsNetId(IQ_stComPortIn.stInfoData.stADSNetId) ,
						nSlaveAddr:=IQ_stComPortIn.stInfoData.nADSPort,

						nSubIndex:=nSubIndex,
						nIndex:=nIndex,

						pSrcBuf:=ADR(bBuffer),
						cbBufLen:=SIZEOF(bBuffer),
						bExecute:=NOT fbEcCoWrite.bBusy,
						tTimeout:=T#3s);

				4:  (* XON/XOFF rx *)
					nIndex:=16#4075;
					nSubIndex:=3;

					IF I_pOptions^.nHandshake = HANDSHAKE_XONXOFF THEN
						bBuffer:=TRUE;
					ELSE
						bBuffer:=FALSE;
					END_IF

					fbEcCoWrite(
						sNetId:=F_CreateAmsNetId(IQ_stComPortIn.stInfoData.stADSNetId) ,
						nSlaveAddr:=IQ_stComPortIn.stInfoData.nADSPort,

						nSubIndex:=nSubIndex,
						nIndex:=nIndex,

						pSrcBuf:=ADR(bBuffer),
						cbBufLen:=SIZEOF(bBuffer),
						bExecute:=NOT fbEcCoWrite.bBusy,
						tTimeout:=T#3s);
			END_CASE

			IF fbEcCoWrite.bBusy = FALSE THEN
				IF fbEcCoWrite.bError = TRUE THEN
					Q_nConfigPortErrorId:=UDINT_TO_INT(fbEcCoWrite.nErrId);
					IQ_stComFlags.bConfigFlag:=FALSE;
				ELSE
					IF nConfigState < 4 THEN
						nConfigState:=nConfigState+1;
					ELSE
						IQ_stComFlags.bConfigFlag:=FALSE;
					END_IF
				END_IF

				IF IQ_stComFlags.bConfigFlag=FALSE THEN
					nConfigState:=0;
				END_IF
			END_IF

		E_ComPortHardware.cComportKL:
			CASE I_pOptions^.eComPortBytes OF
				E_ComPortKlemmenBytes.cComport3Bytes:
					stComPortKL6configuration(Execute :=NOT stComPortKL6configuration.Busy,
						Mode  := SERIALLINEMODE_KL6_3B_ALTERNATIVE,
						Baudrate:= I_pOptions^.nBaudrate,
						NoDatabits:= UDINT_TO_BYTE(I_pOptions^.nDatenbits),
						Parity:= I_pOptions^.nParitaet,
						Stopbits:= UDINT_TO_BYTE(I_pOptions^.nStopbits),
						Handshake:= I_pOptions^.nHandshake,
						pCOMin:= ADR(IQ_stComPortIn.stKlemmeIn3B),
						pCOMout:= ADR(IQ_stComPortOut.stKlemmeOut3B),
						SizeComIn := SIZEOF(IQ_stComPortIn.stKlemmeIn3B));

					IF 	stComPortKL6configuration.Busy = FALSE
						OR stComPortKL6configuration.Error
					THEN
						Q_nConfigPortErrorId:=stComPortKL6configuration.ErrorId;
						IQ_stComFlags.bConfigFlag:=FALSE;
					END_IF

				E_ComPortKlemmenBytes.cComport5Bytes:
					stComPortKL6configuration(Execute:=NOT stComPortKL6configuration.Busy ,
						Mode  := SERIALLINEMODE_KL6_5B_STANDARD,
						Baudrate:= UINT_TO_UDINT(I_pOptions^.nBaudrate),
						NoDatabits:= UDINT_TO_BYTE(I_pOptions^.nDatenbits),
						Parity:= I_pOptions^.nParitaet,
						Stopbits:= UDINT_TO_BYTE(I_pOptions^.nStopbits),
						Handshake:= I_pOptions^.nHandshake,
						pCOMin:= ADR(IQ_stComPortIn.stKlemmeIn5B),
						pCOMout:= ADR(IQ_stComPortOut.stKlemmeOut5B),
						SizeComIn := SIZEOF(IQ_stComPortIn.stKlemmeIn5B) );

					IF 	stComPortKL6configuration.Busy = FALSE
						OR stComPortKL6configuration.Error
					THEN
						Q_nConfigPortErrorId:=stComPortKL6configuration.ErrorId;
						IQ_stComFlags.bConfigFlag:=FALSE;
					END_IF

				E_ComPortKlemmenBytes.cComport22Bytes:
					stComPortKL6configuration(Execute:=NOT stComPortKL6configuration.Busy ,
						Mode  := SERIALLINEMODE_KL6_22B_STANDARD,
						Baudrate:= UDINT_TO_UINT(I_pOptions^.nBaudrate),
						NoDatabits:= UDINT_TO_BYTE(I_pOptions^.nDatenbits),
						Parity:= I_pOptions^.nParitaet,
						Stopbits:= UDINT_TO_BYTE(I_pOptions^.nStopbits),
						Handshake:= I_pOptions^.nHandshake,
						pCOMin:= ADR(IQ_stComPortIn.stKlemmeIn22B),
						pCOMout:= ADR(IQ_stComPortOut.stKlemmeOut22B),
						SizeComIn := SIZEOF(IQ_stComPortIn.stKlemmeIn22B) );

					IF 	stComPortKL6configuration.Busy = FALSE
						OR stComPortKL6configuration.Error
					THEN
						Q_nConfigPortErrorId:=stComPortKL6configuration.ErrorId;
						IQ_stComFlags.bConfigFlag:=FALSE;
					END_IF

			END_CASE
	END_CASE;

	IF IQ_stComFlags.bConfigFlag=FALSE THEN
		(* Einmal nach beenden der Klemmenkonfiguration *)
		Q_stOptionsIntern.tTimeTimeout:=UDINT_TO_TIME(I_pOptions^.nTimeout);


		Q_stOptionsIntern.nLenPrefix:=0;
		Q_stOptionsIntern.sPrefix:='';

		Q_stOptionsIntern.nPrefix:=UDINT_TO_BYTE(I_pOptions^.nPrefix);
		IF Q_stOptionsIntern.nPrefix > 0 THEN
			Q_stOptionsIntern.nLenPrefix:=Q_stOptionsIntern.nLenPrefix+1;
			Q_stOptionsIntern.sPrefix:=CONCAT(Q_stOptionsIntern.sPrefix,CHR(Q_stOptionsIntern.nPrefix));
		END_IF


		Q_stOptionsIntern.nLenSuffix:=0;
		Q_stOptionsIntern.sSuffix:='';

		Q_stOptionsIntern.arrSuffix[1]:=UDINT_TO_BYTE(I_pOptions^.nSuffix1);
		IF Q_stOptionsIntern.arrSuffix[1] > 0 THEN
			Q_stOptionsIntern.nLenSuffix:=Q_stOptionsIntern.nLenSuffix+1;
			Q_stOptionsIntern.sSuffix:=CONCAT(Q_stOptionsIntern.sSuffix,CHR(Q_stOptionsIntern.arrSuffix[1]));
		END_IF

		Q_stOptionsIntern.arrSuffix[2]:=UDINT_TO_BYTE(I_pOptions^.nSuffix2);
		IF Q_stOptionsIntern.arrSuffix[2] > 0 THEN
			Q_stOptionsIntern.nLenSuffix:=Q_stOptionsIntern.nLenSuffix+1;
			Q_stOptionsIntern.sSuffix:=CONCAT(Q_stOptionsIntern.sSuffix,CHR(Q_stOptionsIntern.arrSuffix[2]));

			IF Q_stOptionsIntern.arrSuffix[1] = 0 THEN
				Q_stOptionsIntern.arrSuffix[1]:=Q_stOptionsIntern.arrSuffix[2];
				Q_stOptionsIntern.arrSuffix[2]:=0;
			END_IF
		END_IF


		IF I_pOptions^.nLength > cBufferSize_IntBuffer OR I_pOptions^.nLength = 0 THEN
			Q_stOptionsIntern.nLength:=cBufferSize_IntBuffer;
		ELSE
			Q_stOptionsIntern.nLength:=I_pOptions^.nLength;
		END_IF
	END_IF;
END_IF

END_FUNCTION_BLOCK

// POUs/ComPort_2_0_1_0/FB_ComMain
FUNCTION_BLOCK  FB_ComMain
VAR_INPUT
	// Optionen
	I_pOptions				: POINTER TO ST_ComPortOptions;	// Optionen
	I_pOptionsIntern		: POINTER TO ST_ComPortOptionsIntern;	// Optionen
	
	// Senden
	I_pTxIntBuffer			: POINTER TO ST_ComPortIntBuffer;	//Int Uebergabepuffer
	I_pTxStringBuffer		: POINTER TO ST_ComPortStringBuffer;	// String Uebergabepuffer
	
	I_nTxCount				: INT;	// Anzahl zu sendender Zeichen
	I_eTxProtokoll			: E_ComPortProtokoll;	// Sendenprotokoll
END_VAR

VAR_OUTPUT
	(* Konfiguration *)
	Q_nConfigPortErrorId	: INT;									(* Fehlerrueckmeldung von Konfiguration *)
	
	(* Senden/Empfangen *)
	Q_nComPortErrorId		: INT;									(* Fehlercode beim Senden/Empfangen *)
	Q_sComPortErrorState	: STRING;									(* Status beim Auftreten des Fehlers *)
	
	(* Empfangen *)
	Q_stRxIntBuffer			: ST_ComPortIntBuffer;							(* Int Uebergabepuffer *)
	Q_stRxStringBuffer		: ST_ComPortStringBuffer;						(* String Uebergabepuffer *)
	
	Q_bTimeOut			: BOOL;									(* Timeoutrueckmeldung bei Strignempfang *)
	Q_nRxCount			: INT;									(* Anzahl empfangener Zeichen *)
END_VAR

VAR_IN_OUT
	IQ_stComFlags		: ST_ComPortFlags;
	
	IQ_stRxBuffer		: Tc2_SerialCom.ComBuffer;									(* Interner Empfangspuffer *)
	IQ_stTxBuffer		: Tc2_SerialCom.ComBuffer;									(* Interner Sendepuffer *)
END_VAR

VAR
	fbClearBuffer				: Tc2_SerialCom.ClearComBuffer;
	eProtokoll					: E_ComPortProtokoll;
	                  		
	fTrigRxFlag					: F_TRIG;
	                  		
	rTrigRxFlag					: R_TRIG;
	rTrigTxFlag					: R_TRIG;
	                  		
	rTrigDataReceived			: R_TRIG;
	                  		
	stRxByteBuffer				: Tc2_SerialCom.P3964buffer;
	stTxByteBuffer				: Tc2_SerialCom.P3964buffer;
	                  	
	nRxBufferIndx				: INT;
	nTxBufferIndx				: INT;
	
	
	fbReceiveByteDirect		: Tc2_SerialCom.ReceiveByte;
	fbSendByteDirect			: Tc2_SerialCom.SendByte;
	
	fbReceiveDataBytes		: Tc2_SerialCom.ReceiveData;
	fbSendDataBytes			: Tc2_SerialCom.SendData;
	
	stBarcodeTxStringBuffer	: ST_ComPortStringBuffer;
	
	fbSendReceiveP3964		: Tc2_SerialCom.P3964R;
	fTrigP3964RxBusy			: F_TRIG;
	fTrigP3964TxBusy			: F_TRIG;
	bRxDataReceived			: BOOL;
	
	(* Diagnose *)
	nDiagRxCycleCounter		: UINT;
	nDiagRxErrorCounter		: UINT;
	nDiagRxLastErrorId		: INT;
	nDiagRxDataCounter		: INT;
	
	sDiagMessage				: STRING(50);
	sTmpDiagMessage			: STRING(50);
END_VAR

(* ---------------------------------------------------------------    	*)
(*										*)
(* 	Reset								*)
(*										*)
(*  ---------------------------------------------------------------   	*)
IF IQ_stComFlags.bResetFlag=TRUE
	AND IQ_stComFlags.bConfigFlag = FALSE
THEN
	IQ_stComFlags.bRxFlag:=FALSE;
	IQ_stComFlags.bWaitQuitFlag:=FALSE;
	IQ_stComFlags.bTxFlag:=FALSE;

	IQ_stComFlags.bConfigFlag:=TRUE;

	Q_nComPortErrorId:= 0;
	Q_sComPortErrorState:='';
	Q_bTimeOut:=FALSE;

	nRxBufferIndx:=0;
	WHILE nRxBufferIndx <= cBufferSize_IntBuffer DO
		Q_stRxIntBuffer.arrData[nRxBufferIndx]:=0;
		nRxBufferIndx:=nRxBufferIndx+1;
	END_WHILE

	Q_stRxStringBuffer.sData:='';

	fbClearBuffer(Buffer:=IQ_stRxBuffer);

	fbReceiveDataBytes(Reset:=TRUE ,
		pReceiveData:=ADR(stRxByteBuffer),
		RXbuffer:=IQ_stRxBuffer);

	IQ_stTxBuffer.Count:=0;
	IQ_stTxBuffer.RdIdx:=0;
	IQ_stTxBuffer.WrIdx:=0;
	IQ_stTxBuffer.Error:=0;

	IQ_stRxBuffer.Count:=0;
	IQ_stRxBuffer.RdIdx:=0;
	IQ_stRxBuffer.WrIdx:=0;
	IQ_stRxBuffer.Error:=0;

	(*  Diagnose *)
	nDiagRxCycleCounter:=0;
	nDiagRxErrorCounter:=0;
	nDiagRxLastErrorId:=0;
	nDiagRxDataCounter:=0;

	sTmpDiagMessage:=CONCAT('RxCycle:',UINT_TO_STRING(nDiagRxCycleCounter));
	sTmpDiagMessage:=CONCAT(sTmpDiagMessage,CONCAT(' - RxData:',INT_TO_STRING(nDiagRxDataCounter)));
	sTmpDiagMessage:=CONCAT(sTmpDiagMessage,CONCAT(' - RxError:',UINT_TO_STRING(nDiagRxErrorCounter)));
	sTmpDiagMessage:=CONCAT(sTmpDiagMessage,CONCAT(' - RxErrorId:',INT_TO_STRING(nDiagRxLastErrorId)));
	sDiagMessage:=sTmpDiagMessage;

	IQ_stComFlags.bResetFlag:=FALSE;
END_IF


(* ---------------------------------------------------------------    	*)
(* Allgemein - Senden/Senden P3964			*)
(* ---------------------------------------------------------------    	*)
rTrigRxFlag(CLK:= IQ_stComFlags.bRxFlag);
rTrigTxFlag(CLK:= IQ_stComFlags.bTxFlag);

fTrigRxFlag(CLK:= IQ_stComFlags.bRxFlag);

IF fTrigRxFlag.Q = TRUE THEN
	Q_nComPortErrorId:= 0;
	Q_sComPortErrorState:='';

	Q_bTimeOut:=FALSE;
END_IF


(* ---------------------------------------------------------------    	*)
(*										*)
(* 	Receive								*)
(*										*)
(*  ---------------------------------------------------------------   	*)
IF    IQ_stComFlags.bRxFlag= FALSE
(*    	AND ComFlags.TxFlag = FALSE *)
	AND IQ_stComFlags.bWaitQuitFlag= FALSE
	AND I_pOptions^.nAktiv = 1
	AND IQ_stComFlags.bConfigFlag = FALSE
THEN
	CASE I_pOptions^.eProtokoll OF
		E_ComPortProtokoll.cProtokollNone:;

		E_ComPortProtokoll.cProtokollData:
			fbReceiveDataBytes(
				pPrefix			:= ADR(I_pOptionsIntern^.nPrefix),
				LenPrefix		:= I_pOptionsIntern^.nLenPrefix,
				pSuffix			:= ADR(I_pOptionsIntern^.arrSuffix),
				LenSuffix		:= I_pOptionsIntern^.nLenSuffix,

				Timeout			:= I_pOptionsIntern^.tTimeTimeout,
				Reset				:= FALSE ,

				pReceiveData	:= ADR(stRxByteBuffer),
				SizeReceiveData:= INT_TO_UDINT(I_pOptionsIntern^.nLength),
				RXbuffer			:= IQ_stRxBuffer);

			Q_nComPortErrorId := fbReceiveDataBytes.Error;
			IF Q_nComPortErrorId <> 0 THEN
				Q_nRxCount:=0;
				IQ_stComFlags.bRxFlag := TRUE;
			ELSE
				rTrigDataReceived(CLK:=fbReceiveDataBytes.DataReceived);
				IF rTrigDataReceived.Q THEN
					Q_nRxCount:= UDINT_TO_INT(fbReceiveDataBytes.LenReceiveData);
					nRxBufferIndx:=0;
					WHILE     nRxBufferIndx < Q_nRxCount
						AND nRxBufferIndx <= cBufferSize_IntBuffer
					DO
						Q_stRxIntBuffer.arrData[nRxBufferIndx]:=stRxByteBuffer.D[nRxBufferIndx];
						nRxBufferIndx:=nRxBufferIndx+1;
					END_WHILE

					Q_bTimeOut:= fbReceiveDataBytes.RxTimeout;
					IQ_stComFlags.bRxFlag := TRUE;
				END_IF
			END_IF

		E_ComPortProtokoll.cProtokollDirect:
			fbReceiveByteDirect(RXbuffer:=IQ_stRxBuffer);
			Q_nComPortErrorId := fbReceiveByteDirect.Error;
			IF Q_nComPortErrorId <> 0 THEN
				Q_nRxCount:=0;
				IQ_stComFlags.bRxFlag:=TRUE;
			ELSE
				IF fbReceiveByteDirect.ByteReceived = TRUE THEN
					Q_nRxCount:=0;
					nRxBufferIndx:=0;
					WHILE fbReceiveByteDirect.ByteReceived = TRUE
						AND  nRxBufferIndx <= cBufferSize_IntBuffer
						AND Q_nComPortErrorId = 0
					DO
						Q_stRxIntBuffer.arrData[nRxBufferIndx]:=fbReceiveByteDirect.ReceivedByte;
						Q_nRxCount:=Q_nRxCount +1;

						nRxBufferIndx:=nRxBufferIndx+1;
						IF nRxBufferIndx <= cBufferSize_IntBuffer  THEN
							fbReceiveByteDirect(RXbuffer:=IQ_stRxBuffer);
						END_IF
					END_WHILE

					IQ_stComFlags.bRxFlag:=TRUE;
				END_IF
			END_IF

		E_ComPortProtokoll.cProtokollBarcode:
			fbReceiveDataBytes(pPrefix:=ADR(I_pOptionsIntern^.nPrefix),
				LenPrefix:=I_pOptionsIntern^.nLenPrefix,
				pSuffix:=ADR(I_pOptionsIntern^.arrSuffix),
				LenSuffix:=I_pOptionsIntern^.nLenSuffix,

				Timeout:= I_pOptionsIntern^.tTimeTimeout,
				Reset:=FALSE ,

				pReceiveData:=ADR(Q_stRxStringBuffer),
				SizeReceiveData:=SIZEOF(Q_stRxStringBuffer)-1,
				RXbuffer:=IQ_stRxBuffer);

			Q_nComPortErrorId := fbReceiveDataBytes.Error;
			IF Q_nComPortErrorId <> 0 THEN
				Q_nRxCount:=0;
				IQ_stComFlags.bRxFlag:=TRUE;
			ELSE
				rTrigDataReceived(CLK:=fbReceiveDataBytes.DataReceived);

				IF rTrigDataReceived.Q THEN
					Q_nRxCount	:=UDINT_TO_INT(fbReceiveDataBytes.LenReceiveData);
					IF Q_nRxCount <= cBufferSize_StringBuffer THEN
						Q_stRxStringBuffer.sData:=LEFT(Q_stRxStringBuffer.sData,Q_nRxCount);
					ELSE
						Q_stRxStringBuffer.sData:=LEFT(Q_stRxStringBuffer.sData,cBufferSize_StringBuffer);
					END_IF
					Q_stRxStringBuffer:= F_ComReceiveBarcode(ADR(Q_stRxStringBuffer),I_pOptionsIntern);
					Q_nRxCount:=LEN(Q_stRxStringBuffer.sData);

					Q_bTimeOut:= fbReceiveDataBytes.RxTimeout;
					IQ_stComFlags.bRxFlag := TRUE;
				END_IF;
			END_IF
	END_CASE

	(* Empfang Oberflaeche *)
	IF	IQ_stComFlags.bRxFlag= TRUE
		AND I_pOptions^.nCommVB = 1
	THEN
		IQ_stComFlags.bWaitQuitFlag:=TRUE;
	END_IF
END_IF


(* -----------------------------------------------------------------  	*)
(*										*)
(* 	Send								*)
(*										*)
(*  ----------------------------------------------------------------- 	*)
IF 	IQ_stComFlags.bTxFlag = TRUE
(*	AND ComFlags.RxFlag= FALSE *)
	AND I_pOptions^.nAktiv = 1
	AND IQ_stComFlags.bConfigFlag = FALSE
THEN
	IF I_eTxProtokoll <> E_ComPortProtokoll.cProtokollNone THEN
		eProtokoll := I_eTxProtokoll;
	ELSE
		eProtokoll := I_pOptions^.eProtokoll;
	END_IF

	CASE eProtokoll OF
		E_ComPortProtokoll.cProtokollNone:;

		E_ComPortProtokoll.cProtokollData:
			IF rTrigTxFlag.Q = TRUE  THEN
				Q_nComPortErrorId := 0;

				nTxBufferIndx:=0;
				WHILE     nTxBufferIndx < I_nTxCount
					AND nTxBufferIndx <= cBufferSize_IntBuffer
				DO
					stTxByteBuffer.D[nTxBufferIndx]:=UINT_TO_BYTE(I_pTxIntBuffer^.arrData[nTxBufferIndx]);
					nTxBufferIndx:=nTxBufferIndx+1;
				END_WHILE
			END_IF

			fbSendDataBytes(
				pSendData:= ADR(stTxByteBuffer),
				Length	:= INT_TO_UDINT(I_nTxCount),
				TXbuffer	:= IQ_stTxBuffer);

			Q_nComPortErrorId := fbSendDataBytes.Error;
			IF Q_nComPortErrorId <> 0 THEN
				I_eTxProtokoll := E_ComPortProtokoll.cProtokollNone;
				IQ_stComFlags.bTxFlag := FALSE;
			ELSE
				IF fbSendDataBytes.Busy = FALSE  THEN
					I_eTxProtokoll := E_ComPortProtokoll.cProtokollNone;
					IQ_stComFlags.bTxFlag := FALSE;
				END_IF
			END_IF

		E_ComPortProtokoll.cProtokollDirect:
			IF rTrigTxFlag.Q = TRUE  THEN
				Q_nComPortErrorId := 0;

				nTxBufferIndx := 0;
				IF I_nTxCount > cBufferSize_IntBuffer THEN
					I_nTxCount := cBufferSize_IntBuffer;
				END_IF
			END_IF

			IF fbSendByteDirect.Busy = FALSE THEN
				WHILE     nTxBufferIndx < I_nTxCount
					AND Q_nComPortErrorId = 0
					AND fbSendByteDirect.Busy = FALSE
				DO
					fbSendByteDirect(SendByte:=UINT_TO_BYTE(I_pTxIntBuffer^.arrData[nTxBufferIndx]),
						TXbuffer:=IQ_stTxBuffer);
					Q_nComPortErrorId := fbSendByteDirect.Error;

					nTxBufferIndx:=nTxBufferIndx+1;
				END_WHILE
			END_IF

			IF (nTxBufferIndx >= I_nTxCount  AND fbSendByteDirect.Busy = FALSE ) OR Q_nComPortErrorId <> 0 THEN
				I_eTxProtokoll := E_ComPortProtokoll.cProtokollNone;
				IQ_stComFlags.bTxFlag := FALSE;
			END_IF

		E_ComPortProtokoll.cProtokollBarcode:
			IF rTrigTxFlag.Q = TRUE  THEN
				Q_nComPortErrorId := 0;
				stBarcodeTxStringBuffer:= F_ComSendBarcode(I_pTxStringBuffer,I_pOptionsIntern);
			END_IF

			fbSendDataBytes(pSendData:=ADR(stBarcodeTxStringBuffer),
				Length:=INT_TO_BYTE(LEN(stBarcodeTxStringBuffer.sData)),
				TXbuffer:=IQ_stTxBuffer);

			Q_nComPortErrorId := fbSendDataBytes.Error;
			IF Q_nComPortErrorId <> 0 THEN
				I_eTxProtokoll := E_ComPortProtokoll.cProtokollNone;
				IQ_stComFlags.bTxFlag := FALSE;
			ELSE
				IF fbSendDataBytes.Busy = FALSE  THEN
					I_eTxProtokoll := E_ComPortProtokoll.cProtokollNone;
					IQ_stComFlags.bTxFlag := FALSE;
				END_IF
			END_IF
	END_CASE
END_IF


(* ---------------------------------------------------------------    	*)
(*										*)
(* 	Receive/Sende P3964   				*)
(*										*)
(*  ---------------------------------------------------------------   *)
IF I_pOptions^.eProtokoll = E_ComPortProtokoll.cProtokollP3964 THEN
	IF I_pOptions^.nAktiv = 1
		AND IQ_stComFlags.bConfigFlag = FALSE
	THEN
		IF rTrigTxFlag.Q THEN
			(* Senden starten *)
			IF I_nTxCount > cBufferSize_IntBuffer THEN
				I_nTxCount := cBufferSize_IntBuffer;
			END_IF

			Q_nComPortErrorId := 0;

			nTxBufferIndx:=0;
			WHILE nTxBufferIndx < I_nTxCount DO
				stTxByteBuffer.D[nTxBufferIndx]:=UINT_TO_BYTE(I_pTxIntBuffer^.arrData[nTxBufferIndx]);
				nTxBufferIndx:=nTxBufferIndx+1;
			END_WHILE
		END_IF

		(* Senden/Empfangen *)
		fbSendReceiveP3964(
			TXstart:=fbSendReceiveP3964.TXbusy=FALSE  AND fbSendReceiveP3964.RXbusy=FALSE   AND IQ_stComFlags.bTxFlag,
			RXstart:=NOT fbSendReceiveP3964.Busy,
			TXcount:=I_nTxCount,
			Priority:=FALSE ,
			TXdata:=stTxByteBuffer ,
			RXdata:=stRxByteBuffer,
			TXbuffer:=IQ_stTxBuffer,
			RXbuffer:=IQ_stRxBuffer);


		fTrigP3964TxBusy(CLK:=  fbSendReceiveP3964.TXbusy);
		IF fTrigP3964TxBusy.Q THEN
			(* Senden abgeschlossen *)
			IF  fbSendReceiveP3964.Error = FALSE THEN
				Q_nComPortErrorId:= 0;
				Q_sComPortErrorState:='';
			ELSE
				Q_nComPortErrorId:=fbSendReceiveP3964.ErrorId;
				Q_sComPortErrorState:=fbSendReceiveP3964.ErrorState;
			END_IF

			I_eTxProtokoll := E_ComPortProtokoll.cProtokollNone;
			IQ_stComFlags.bTxFlag := FALSE;
		END_IF

		fTrigP3964RxBusy(CLK:=  fbSendReceiveP3964.RXbusy);
		IF fTrigP3964RxBusy.Q THEN
			(* Empfang abgeschlossen *)
			IF bRxDataReceived = TRUE THEN
				(* Daten noch nicht uebernommen *)
				Q_nComPortErrorId:=99;
				Q_sComPortErrorState:='RxFlag';
			ELSE
				IF  fbSendReceiveP3964.Error = FALSE THEN
					Q_nComPortErrorId:= 0;
					Q_sComPortErrorState:='';
				ELSE
					Q_nComPortErrorId:=fbSendReceiveP3964.ErrorId;
					Q_sComPortErrorState:=fbSendReceiveP3964.ErrorState;
				END_IF

				bRxDataReceived:=TRUE;
			END_IF
		END_IF


		IF   bRxDataReceived = TRUE
			AND IQ_stComFlags.bRxFlag = FALSE
			AND IQ_stComFlags.bWaitQuitFlag= FALSE
		THEN
			(* Daten ausgelesen *)
			Q_nRxCount:=fbSendReceiveP3964.RxCount;

			nRxBufferIndx:=0;
			WHILE     nRxBufferIndx < Q_nRxCount
				AND nRxBufferIndx <= cBufferSize_IntBuffer
			DO
				Q_stRxIntBuffer.arrData[nRxBufferIndx]:=stRxByteBuffer.D[nRxBufferIndx];
				nRxBufferIndx:=nRxBufferIndx+1;
			END_WHILE

			IF  fbSendReceiveP3964.Error = TRUE THEN
				Q_nComPortErrorId:=fbSendReceiveP3964.ErrorId;
				Q_sComPortErrorState:=fbSendReceiveP3964.ErrorState;
			END_IF

			bRxDataReceived:=FALSE;
			IQ_stComFlags.bRxFlag := TRUE;
			IF I_pOptions^.nCommVB = 1 THEN
				IQ_stComFlags.bWaitQuitFlag:=TRUE;
			END_IF
		END_IF
	END_IF
END_IF


(* ---------------------------------------------------------------    	*)
(* Allgemein - Senden/Senden P3964*)
(* ---------------------------------------------------------------    	*)
fTrigRxFlag(CLK:= IQ_stComFlags.bRxFlag);

rTrigRxFlag(CLK:= IQ_stComFlags.bRxFlag);
rTrigTxFlag(CLK:= IQ_stComFlags.bTxFlag);


(* ---------------------------------------------------------------    	*)
(*										*)
(* 	Diagnose                          					*)
(*										*)
(*  ---------------------------------------------------------------   	*)
IF rTrigRxFlag.Q THEN
	(* Diagnoseauswertung  Empfang *)
	IF nDiagRxCycleCounter >= 9999
		OR nDiagRxErrorCounter >= 9999
		OR nDiagRxDataCounter + Q_nRxCount >= 9999
	THEN
		nDiagRxCycleCounter:=0;
		nDiagRxErrorCounter:=0;
		nDiagRxDataCounter:=0;
	END_IF

	nDiagRxCycleCounter:=nDiagRxCycleCounter+1;
	IF Q_nComPortErrorId = 0 THEN
		nDiagRxDataCounter:=nDiagRxDataCounter + Q_nRxCount;
	ELSE
		nDiagRxErrorCounter:=nDiagRxErrorCounter+1;
		nDiagRxLastErrorId:=Q_nComPortErrorId;
	END_IF

	sTmpDiagMessage:=CONCAT('RxCycle:',UINT_TO_STRING(nDiagRxCycleCounter));
	sTmpDiagMessage:=CONCAT(sTmpDiagMessage,CONCAT(' - RxData:',INT_TO_STRING(nDiagRxDataCounter)));
	sTmpDiagMessage:=CONCAT(sTmpDiagMessage,CONCAT(' - RxError:',UINT_TO_STRING(nDiagRxErrorCounter)));
	sTmpDiagMessage:=CONCAT(sTmpDiagMessage,CONCAT(' - RxErrorId:',INT_TO_STRING(nDiagRxLastErrorId)));
	sDiagMessage:=sTmpDiagMessage;
END_IF

END_FUNCTION_BLOCK

// POUs/ComPort_2_0_1_0/FB_ComPortOld
FUNCTION_BLOCK FB_ComPortOld
VAR_INPUT
	I_stOptions				: ST_ComPortOptions;
	I_stComFlags			: ST_ComPortFlags;

	I_stTxIntBuffer		: ST_ComPortIntBuffer;		(* Int Uebergabepuffer *)
	I_stTxStringBuffer	: ST_ComPortStringBuffer;	(* String Uebergabepuffer *)

	I_nTxCount				: INT;				(* Anzahl zu sendender Zeichen *)
	I_eTxProtokoll			: E_ComPortProtokoll;		(* Sendenprotokoll *)
END_VAR

VAR
	stComPortIn 	AT %I*	: ST_ComPortInData;
	stComPortOut 	AT %Q*	: ST_ComPortOutData;

	fbComBackgroundFunction: FB_ComBackground;

	fbComConfigFunction		: FB_ComConfig;
	fbComMainFunction			: FB_ComMain;

	stRxBuffer					: Tc2_SerialCom.ComBuffer;			(* Interner Empfangspuffer *)
	stTxBuffer					: Tc2_SerialCom.ComBuffer;			(* Interner Sendepuffer *)

	stOptionsIntern			: ST_ComPortOptionsIntern;
                        	
	nConfigPortErrorId		: INT;
                        	
	nComPortErrorId			: INT;				(* Fehlercode beim Senden/Empfangen *)
	sComPortErrorState		: STRING;				(* Status beim Auftreten des Fehlers *)
                        	
	stRxIntBuffer				: ST_ComPortIntBuffer;		(* Int Uebergabepuffer *)
	stRxStringBuffer			: ST_ComPortStringBuffer;	(* String Uebergabepuffer  *)
                        	
	bRxTimeout					: BOOL;				(* Timeoutrueckmeldung bei Strignempfang *)
	nRxCount						: INT;				(* Anzahl empfangener Zeichen *)
END_VAR

(* Schnittstellenkonfiguration *)
fbComConfigFunction(
I_pOptions:= ADR(I_stOptions),

IQ_stComPortIn:=stComPortIn,
IQ_stComPortOut:=stComPortOut,

IQ_stComFlags:= I_stComFlags);

stOptionsIntern:=fbComConfigFunction.Q_stOptionsIntern;
nConfigPortErrorId:=fbComConfigFunction.Q_nConfigPortErrorId;


(* Zentrale Kommunikationsfunktion *)
fbComMainFunction(
I_pOptions:=ADR(I_stOptions) ,
I_pOptionsIntern:= ADR(stOptionsIntern),
I_pTxIntBuffer:=ADR(I_stTxIntBuffer) ,
I_pTxStringBuffer:=ADR(I_stTxStringBuffer),
I_nTxCount:=I_nTxCount ,
I_eTxProtokoll:=I_eTxProtokoll ,
IQ_stComFlags:=I_stComFlags ,
IQ_stRxBuffer:=stRxBuffer ,
IQ_stTxBuffer:=stTxBuffer );


nConfigPortErrorId:=fbComMainFunction.Q_nConfigPortErrorId;

nComPortErrorId:=fbComMainFunction.Q_nComPortErrorId;
sComPortErrorState:=fbComMainFunction.Q_sComPortErrorState;

stRxIntBuffer:=fbComMainFunction.Q_stRxIntBuffer;
stRxStringBuffer:=fbComMainFunction.Q_stRxStringBuffer;
bRxTimeout:=fbComMainFunction.Q_bTimeOut;
nRxCount:=fbComMainFunction.Q_nRxCount;

END_FUNCTION_BLOCK

// POUs/ComPort_3_0_1_0/FB_ComPort
// Steuern, konfigurieren, senden und empfangen mit und über eine serielle Klemme. Um die Klemme konfigurieren zu können muss die ADS-NetId aus der Input-Struktur verknüpft werden. Die seriellen EL-Klemme haben diesen Eingang auf jeden Fall.
FUNCTION_BLOCK FB_ComPort
VAR_OUTPUT
	Q_stMeldungen					: ST_MeldComPort;		// Meldestruktur für Avalon
END_VAR
VAR
	stComPortIn 	AT %I*	: ST_ComPortInData;	// Hardwarevariable
	stComPortOut 	AT %Q*	: ST_ComPortOutData;	// Hardwarevariable
	
	stOptionsIntern			: ST_ComPortOptionsIntern;	// Bytestreamkonfiguration
	stOptions					: ST_ComPortOptions;	// Schnittstellenkonfiguration

	stRxIntBuffer				: ST_ComPortIntBuffer;	// Int Uebergabepuffer
	stRxStringBuffer			: ST_ComPortStringBuffer;	// String Uebergabepuffer
	
	stConfigResult				: ST_MethodResult;
	stReceiveResult			: ST_MethodResult;
	stSendResult				: ST_MethodResult;	// Wird innerhalb der Methode beschrieben, da die Methode nicht intern aufgerufen wird, wie die Recieve-Methode
	
// ccl_Main	
	bStartPLC					: BOOL;	// Erster Zyklus. SPS Startet
	bWartenAufVBA_HMI			: BOOL;	// Warten, bis die VBA-HMI die neuen Daten ausgelesen hat.

	// Diagnose
	nDiagRxCycleCounter		: UINT;
	nDiagRxErrorCounter		: UINT;
	nDiagRxLastErrorId		: INT;
	nDiagRxDataCounter		: INT;
	
	sDiagMessage				: STRING(50);
	sTmpDiagMessage			: STRING(50);

// ccl_Background
	fbPCComPortControl				: Tc2_SerialCom.SerialLineControl;
	fbKlemmeComPortControl3Bytes 	: Tc2_SerialCom.SerialLineControl;
	fbKlemmeComPortControl5Bytes 	: Tc2_SerialCom.SerialLineControl;
	fbKlemmeComPortControl22Bytes	: Tc2_SerialCom.SerialLineControl;
	
// nccl_Config
	fbComPortKL6configuration	: Tc2_SerialCom.KL6configuration;

	fbEcCoWrite				: Tc2_EtherCAT.FB_EcCoESdoWrite;

	nIndex					: WORD;
	nSubIndex				: BYTE;

	nWordBuffer				: WORD;
	bBuffer					: BOOL;

	nConfigState			: INT;
	nTmpVar					: UINT;
	
// nccl_Send
	stTxBuffer				: Tc2_SerialCom.ComBuffer;	//Interner Sendepuffer
	
// ccl_Receive
	stRxBuffer				: Tc2_SerialCom.ComBuffer;	//Interner Empfangspuffer
	stRxByteBuffer			: Tc2_SerialCom.P3964buffer;	// Ist eigentlich nur ein Byte-Array
	
	fbReceiveByteDirect	: Tc2_SerialCom.ReceiveByte;
	fbReceiveDataBytes	: Tc2_SerialCom.ReceiveData;

	RxFlagFallingEdge		: Tc2_Standard.F_TRIG;
	RxFlagRisingEdge		: Tc2_Standard.R_TRIG;
	
	bRxTimeout				: BOOL;	// Timeoutrückmeldung bei Stringempfang *)
	nRxCount					: INT;	// Anzahl empfangener Zeichen
	bNeueDatenEmpfangen	: BOOL;	// es sind neue Daten zum auslesen vorhanden.
END_VAR

// Zentrale Kommunikationsfunktion
ccl_Main();

METHOD PUBLIC ccl_Backround : BOOL	// bei KL-Klemmen in einer 3ms Task aufrufen. Bei EL-Klemmen ist das glaube ich nicht so wichtig.
IF stOptions.nAktiv = 1
	AND NOT stConfigResult.bBusy 
THEN
	CASE stOptions.ePort OF
		E_ComPortHardware.cComportPc:
			fbPCComPortControl(
				Mode  		:= SERIALLINEMODE_PC_COM_PORT,
				pCOMin		:= ADR(stComPortIn.stPCIn) ,
				pCOMout		:= ADR(stComPortOut.stPCOut) ,
				SizeComIn	:= UINT_TO_INT(SIZEOF(stComPortIn.stPCIn)),
				TxBuffer		:= stTxBuffer ,
				RxBuffer		:= stRxBuffer
			);

		E_ComPortHardware.cComportKL,E_ComPortHardware.cComportEL:
			CASE stOptions.eComPortBytes OF
				E_ComPortKlemmenBytes.cComport3Bytes:
					fbKlemmeComPortControl3Bytes(
						Mode  		:= SERIALLINEMODE_KL6_3B_ALTERNATIVE,
						pCOMin		:= ADR(stComPortIn.stKlemmeIn3B) ,
						pCOMout		:= ADR(stComPortOut.stKlemmeOut3B) ,
						SizeComIn	:= UINT_TO_INT(SIZEOF(stComPortIn.stKlemmeIn3B)),
						TxBuffer		:= stTxBuffer ,
						RxBuffer		:= stRxBuffer
					);

				E_ComPortKlemmenBytes.cComport5Bytes:
					fbKlemmeComPortControl5Bytes(
						Mode  		:= SERIALLINEMODE_KL6_5B_STANDARD,
						pCOMin		:= ADR(stComPortIn.stKlemmeIn5B) ,
						pCOMout		:= ADR(stComPortOut.stKlemmeOut5B) ,
						SizeComIn	:= UINT_TO_INT(SIZEOF(stComPortIn.stKlemmeIn5B)),
						TxBuffer		:= stTxBuffer ,
						RxBuffer		:= stRxBuffer
					);

				E_ComPortKlemmenBytes.cComport22Bytes:
					fbKlemmeComPortControl22Bytes(
						Mode  		:= SERIALLINEMODE_KL6_22B_STANDARD,
						pCOMin		:= ADR(stComPortIn.stKlemmeIn22B) ,
						pCOMout		:= ADR(stComPortOut.stKlemmeOut22B) ,
						SizeComIn	:= UINT_TO_INT(SIZEOF(stComPortIn.stKlemmeIn22B)),
						TxBuffer		:= stTxBuffer ,
						RxBuffer		:= stRxBuffer
					);
			END_CASE
	END_CASE;
END_IF
END_METHOD

METHOD PUBLIC ccl_Main : BOOL	// Muss zyklisch in der normalen Task aufgerufen werden. Wahlweise kann auch der FB aufgerufen werden. Hat den gleichen Effekt.
// Schnittstellenkonfiguration
IF NOT bStartPLC
THEN
	stConfigResult := nccl_Config();
	IF stConfigResult.bDone
	THEN
		bStartPLC	:= TRUE;
	END_IF
END_IF


// Daten Empfangen
RxFlagRisingEdge(CLK:= bNeueDatenEmpfangen);
RxFlagFallingEdge(CLK:= bNeueDatenEmpfangen);
IF RxFlagFallingEdge.Q
THEN
	bRxTimeout				:= FALSE;
END_IF

stReceiveResult	:= ccl_Receive();

// Diagnose der Empfangenen Daten
IF RxFlagRisingEdge.Q
THEN
	(* Diagnoseauswertung  Empfang *)
	IF nDiagRxCycleCounter >= 9999
		OR nDiagRxErrorCounter >= 9999
		OR nDiagRxDataCounter + nRxCount >= 9999
	THEN
		nDiagRxCycleCounter	:= 0;
		nDiagRxErrorCounter	:= 0;
		nDiagRxDataCounter	:= 0;
	END_IF

	nDiagRxCycleCounter	:= nDiagRxCycleCounter+1;
	
	IF stReceiveResult.nErrorId = 0
	THEN
		nDiagRxDataCounter	:= nDiagRxDataCounter + nRxCount;
	ELSE
		nDiagRxErrorCounter	:= nDiagRxErrorCounter+1;
		nDiagRxLastErrorId	:= stReceiveResult.nErrorId;
	END_IF

	sTmpDiagMessage	:= CONCAT('RxCycle:', UINT_TO_STRING(nDiagRxCycleCounter));
	sTmpDiagMessage	:= CONCAT(sTmpDiagMessage, CONCAT(' - RxData:', INT_TO_STRING(nDiagRxDataCounter)));
	sTmpDiagMessage	:= CONCAT(sTmpDiagMessage, CONCAT(' - RxError:', UINT_TO_STRING(nDiagRxErrorCounter)));
	sTmpDiagMessage	:= CONCAT(sTmpDiagMessage, CONCAT(' - RxErrorId:', INT_TO_STRING(nDiagRxLastErrorId)));
	sDiagMessage		:= sTmpDiagMessage;
END_IF

ccl_Messages();
END_METHOD

METHOD PRIVATE ccl_Messages : BOOL
VAR_INPUT
END_VAR

// Konfig Meldungen
Q_stMeldungen.bMeldConfig	:=
	NOT bStartplc
	AND stOptions.nAktiv = 1;	// Meldung, wenn die Config nicht fertig ist.

Q_stMeldungen.nConfigError	:=	stConfigResult.nErrorId;
Q_stMeldungen.bMeldConfigError	:=
	stConfigResult.bError
	AND stOptions.nAktiv = 1;	// Meldung bei Fehler wärend der Konfiguration

Q_stMeldungen.bMeldMissingLink	:=
	((stComPortIn.stInfoData.nADSPort = 0)	// Fehler, wenn nicht alle Varablen verküpft sind.
		OR ((stComPortIn.stInfoData.stADSNetId[0]= 0)
			AND (stComPortIn.stInfoData.stADSNetId[1]= 0)
			AND (stComPortIn.stInfoData.stADSNetId[2]= 0)
			AND (stComPortIn.stInfoData.stADSNetId[3]= 0)
			AND (stComPortIn.stInfoData.stADSNetId[4]= 0)
			AND (stComPortIn.stInfoData.stADSNetId[5]= 0)))
	AND stOptions.nAktiv = 1;

// Datenempfang
Q_stMeldungen.nRecieveError	:=	stReceiveResult.nErrorId;
Q_stMeldungen.bMeldRecieveError	:=
	stReceiveResult.bError
	AND stOptions.nAktiv = 1;	// Meldung bei Empfangen von Daten

Q_stMeldungen.tTimeoutZeit	:= stOptionsIntern.tTimeTimeout;
Q_stMeldungen.bMeldRecieveTimeout	:=
	bRxTimeout
	AND stOptions.nAktiv = 1;
	
// Daten senden
Q_stMeldungen.nSendError	:= stSendResult.nErrorId;
Q_stMeldungen.bMeldSendError	:=
	stSendResult.bError
	AND stOptions.nAktiv = 1;
END_METHOD

METHOD INTERNAL ccl_Receive : ST_MethodResult	// Diese Methode muss zyklisch aufgerufen werden.
VAR
	nRxBufferIndx	: INT;
END_VAR
// Daten Empfangen
IF NOT bNeueDatenEmpfangen
	AND NOT bWartenAufVBA_HMI
	AND NOT stConfigResult.bBusy
	AND stOptions.nAktiv = 1
THEN

	ccl_Receive.bBusy	:= TRUE;

	CASE stOptions.eProtokoll OF
		
		E_ComPortProtokoll.cProtokollNone:
			;
			
		E_ComPortProtokoll.cProtokollData:
		
			// Zyklisch auf neue Daten auslesen pollen
			fbReceiveDataBytes(
				pPrefix			:= ADR(stOptionsIntern.sPrefix),
				LenPrefix		:= stOptionsIntern.nLenPrefix,
				pSuffix			:= ADR(stOptionsIntern.sSuffix),
				LenSuffix		:= stOptionsIntern.nLenSuffix,

				Timeout			:= stOptionsIntern.tTimeTimeout,
				Reset				:= FALSE ,

				pReceiveData	:= ADR(stRxByteBuffer),
				SizeReceiveData:= INT_TO_UDINT(stOptionsIntern.nLength),
				RXbuffer			:= stRxBuffer
			);
			
			IF fbReceiveDataBytes.Error <> 0
			THEN	// Fehler beim Datenempfangen
				nRxCount					:= 0;
				bNeueDatenEmpfangen	:= TRUE;
				ccl_Receive.bBusy		:= FALSE;
				ccl_Receive.bDone		:= TRUE;
				ccl_Receive.bError	:= TRUE;
				ccl_Receive.nErrorId	:= fbReceiveDataBytes.Error;
			ELSE
				
				IF fbReceiveDataBytes.DataReceived
				THEN	// Es wurden Daten empfangen.
					nRxCount	:= UDINT_TO_INT(fbReceiveDataBytes.LenReceiveData);
					
					nRxBufferIndx	:=0;
					WHILE nRxBufferIndx < nRxCount
						AND nRxBufferIndx <= cBufferSize_IntBuffer
					DO
						stRxIntBuffer.arrData[nRxBufferIndx]	:= stRxByteBuffer.D[nRxBufferIndx];
						nRxBufferIndx	:=nRxBufferIndx+1;
					END_WHILE

					bRxTimeout	:= fbReceiveDataBytes.RxTimeout;
					bNeueDatenEmpfangen	:= TRUE;
				END_IF
			END_IF

		E_ComPortProtokoll.cProtokollDirect:
		
			// Aufrufen und damit quasi warten bis der Bytestream anfängt.
			fbReceiveByteDirect(RXbuffer	:= stRxBuffer);
			
			IF fbReceiveByteDirect.Error <> 0
			THEN	// Fehler beim Datenempfangen
				nRxCount					:= 0;
				bNeueDatenEmpfangen	:= TRUE;
				ccl_Receive.bBusy		:= FALSE;
				ccl_Receive.bDone		:= TRUE;
				ccl_Receive.bError	:= TRUE;
				ccl_Receive.nErrorId	:= fbReceiveByteDirect.Error;
			ELSE
				IF fbReceiveByteDirect.ByteReceived
				THEN	// Es wurde mindestens ein Datum empfangen. Jetzt so lange auslesen, bis nichts mehr im Buffer ist.
					nRxCount			:= 0;
					nRxBufferIndx	:= 0;
					
					WHILE fbReceiveByteDirect.ByteReceived
						AND nRxBufferIndx <= cBufferSize_IntBuffer
						AND fbReceiveByteDirect.Error = 0
					DO
						stRxIntBuffer.arrData[nRxBufferIndx]	:= fbReceiveByteDirect.ReceivedByte;
						nRxCount	:= nRxCount +1;

						nRxBufferIndx	:= nRxBufferIndx+1;
						IF nRxBufferIndx <= cBufferSize_IntBuffer
						THEN
							fbReceiveByteDirect(RXbuffer	:= stRxBuffer);
						END_IF
						
					END_WHILE

					// Daten sind fertig empfangen
					bNeueDatenEmpfangen	:= TRUE;
					
				END_IF
			END_IF

		E_ComPortProtokoll.cProtokollBarcode:
		
